gfCNCPoint4[7267] = {X 587.5052, Y 48.1018, Z -5.5000, A 0.000, B 0.000, C 0.000 }
gfCNCPoint4[7268] = {X 587.0658, Y 48.8401, Z -5.5000, A 0.000, B 0.000, C 0.000 }
gfCNCPoint4[7269] = {X 586.5368, Y 49.5171, Z -5.5000, A 0.000, B 0.000, C 0.000 }
gfCNCPoint4[7270] = {X 585.9266, Y 50.1220, Z -5.5000, A 0.000, B 0.000, C 0.000 }
gfCNCPoint4[7271] = {X 585.1803, Y 50.6880, Z -5.5000, A 0.000, B 0.000, C 0.000 }
gfCNCPoint4[7272] = {X 584.3634, Y 51.1461, Z -5.5000, A 0.000, B 0.000, C 0.000 }
gfCNCPoint4[7273] = {X 583.3013, Y 51.5442, Z -5.5000, A 0.000, B 0.000, C 0.000 }
gfCNCPoint4[7274] = {X 582.1877, Y 51.7603, Z -5.5000, A 0.000, B 0.000, C 0.000 }
gfCNCPoint4[7275] = {X 581.0538, Y 51.7882, Z -5.5000, A 0.000, B 0.000, C 0.000 }
gfCNCPoint4[7276] = {X 579.9310, Y 51.6273, Z -5.5000, A 0.000, B 0.000, C 0.000 }
gfCNCPoint4[7277] = {X 578.8505, Y 51.2819, Z -5.5000, A 0.000, B 0.000, C 0.000 }
gfCNCPoint4[7278] = {X 577.8425, Y 50.7618, Z -5.5000, A 0.000, B 0.000, C 0.000 }
gfCNCPoint4[7279] = {X 576.9350, Y 50.0813, Z -5.5000, A 0.000, B 0.000, C 0.000 }
gfCNCPoint4[7280] = {X 576.3133, Y 49.4513, Z -5.5000, A 0.000, B 0.000, C 0.000 }
gfCNCPoint4[7281] = {X 575.7786, Y 48.7459, Z -5.5000, A 0.000, B 0.000, C 0.000 }
gfCNCPoint4[7282] = {X 575.3401, Y 47.9770, Z -5.5000, A 0.000, B 0.000, C 0.000 }
gfCNCPoint4[7283] = {X 574.9017, Y 48.7459, Z -5.5000, A 0.000, B 0.000, C 0.000 }
gfCNCPoint4[7284] = {X 574.3670, Y 49.4513, Z -5.5000, A 0.000, B 0.000, C 0.000 }
gfCNCPoint4[7285] = {X 573.7453, Y 50.0813, Z -5.5000, A 0.000, B 0.000, C 0.000 }
gfCNCPoint4[7286] = {X 572.7526, Y 50.8143, Z -5.5000, A 0.000, B 0.000, C 0.000 }
gfCNCPoint4[7287] = {X 571.6437, Y 51.3558, Z -5.5000, A 0.000, B 0.000, C 0.000 }
gfCNCPoint4[7288] = {X 570.4553, Y 51.6880, Z -5.5000, A 0.000, B 0.000, C 0.000 }
gfCNCPoint4[7289] = {X 569.2264, Y 51.8000, Z -5.5000, A 0.000, B 0.000, C 0.000 }
gfCNCPoint4[7290] = {X 562.4443, Y 51.8000, Z -5.5000, A 0.000, B 0.000, C 0.000 }
gfCNCPoint4[7291] = {X 561.2635, Y 51.6967, Z -5.5000, A 0.000, B 0.000, C 0.000 }
gfCNCPoint4[7292] = {X 560.1186, Y 51.3899, Z -5.5000, A 0.000, B 0.000, C 0.000 }
gfCNCPoint4[7293] = {X 559.0443, Y 50.8890, Z -5.5000, A 0.000, B 0.000, C 0.000 }
gfCNCPoint4[7294] = {X 558.0733, Y 50.2091, Z -5.5000, A 0.000, B 0.000, C 0.000 }
gfCNCPoint4[7295] = {X 557.2352, Y 49.3710, Z -5.5000, A 0.000, B 0.000, C 0.000 }
gfCNCPoint4[7296] = {X 556.5553, Y 48.4000, Z -5.5000, A 0.000, B 0.000, C 0.000 }
gfCNCPoint4[7297] = {X 556.0544, Y 47.3257, Z -5.5000, A 0.000, B 0.000, C 0.000 }
gfCNCPoint4[7298] = {X 555.7476, Y 46.1808, Z -5.5000, A 0.000, B 0.000, C 0.000 }
gfCNCPoint4[7299] = {X 555.6443, Y 45.0000, Z -5.5000, A 0.000, B 0.000, C 0.000 }
gfCNCPoint4[7300] = {X 555.6443, Y 44.0662, Z -5.5000, A 0.000, B 0.000, C 0.000 }
gfCNCPoint4[7301] = {X 555.7452, Y 42.9113, Z -5.5000, A 0.000, B 0.000, C 0.000 }
gfCNCPoint4[7302] = {X 556.0400, Y 41.7902, Z -5.5000, A 0.000, B 0.000, C 0.000 }
gfCNCPoint4[7303] = {X 556.5200, Y 40.7350, Z -5.5000, A 0.000, B 0.000, C 0.000 }
gfCNCPoint4[7304] = {X 557.1715, Y 39.7762, Z -5.5000, A 0.000, B 0.000, C 0.000 }
gfCNCPoint4[7305] = {X 557.1715, Y 10.2279, Z -5.5000, A 0.000, B 0.000, C 0.000 }
gfCNCPoint4[7306] = {X 556.5255, Y 9.2818, Z -5.5000, A 0.000, B 0.000, C 0.000 }
gfCNCPoint4[7307] = {X 556.0475, Y 8.2407, Z -5.5000, A 0.000, B 0.000, C 0.000 }
gfCNCPoint4[7308] = {X 555.7510, Y 7.1341, Z -5.5000, A 0.000, B 0.000, C 0.000 }
gfCNCPoint4[7309] = {X 555.6446, Y 5.9935, Z -5.5000, A 0.000, B 0.000, C 0.000 }
gfCNCPoint4[7310] = {X 555.6443, Y 5.0000, Z -5.5000, A 0.000, B 0.000, C 0.000 }
gfCNCPoint4[7311] = {X 555.6452, Y 4.8909, Z -5.5000, A 0.000, B 0.000, C 0.000 }
gfCNCPoint4[7312] = {X 555.6478, Y 4.7819, Z -5.5000, A 0.000, B 0.000, C 0.000 }
gfCNCPoint4[7313] = {X 555.8079, Y 3.5174, Z -5.5000, A 0.000, B 0.000, C 0.000 }
gfCNCPoint4[7314] = {X 556.2012, Y 2.3049, Z -5.5000, A 0.000, B 0.000, C 0.000 }
gfCNCPoint4[7315] = {X 358.2599, Y 2.3049, Z -5.5000, A 0.000, B 0.000, C 0.000 }
gfCNCPoint4[7316] = {X 360.1211, Y 3.4745, Z -5.5000, A 0.000, B 0.000, C 0.000 }
gfCNCPoint4[7317] = {X 361.8537, Y 4.8274, Z -5.5000, A 0.000, B 0.000, C 0.000 }
gfCNCPoint4[7318] = {X 363.4396, Y 6.3495, Z -5.5000, A 0.000, B 0.000, C 0.000 }
gfCNCPoint4[7319] = {X 363.8248, Y 6.7699, Z -5.5000, A 0.000, B 0.000, C 0.000 }
gfCNCPoint4[7320] = {X 364.1987, Y 7.2003, Z -5.5000, A 0.000, B 0.000, C 0.000 }
gfCNCPoint4[7321] = {X 365.5801, Y 8.9956, Z -5.5000, A 0.000, B 0.000, C 0.000 }
gfCNCPoint4[7322] = {X 366.7977, Y 10.9058, Z -5.5000, A 0.000, B 0.000, C 0.000 }
gfCNCPoint4[7323] = {X 367.8422, Y 12.9160, Z -5.5000, A 0.000, B 0.000, C 0.000 }
gfCNCPoint4[7324] = {X 368.7052, Y 15.0104, Z -5.5000, A 0.000, B 0.000, C 0.000 }
gfCNCPoint4[7325] = {X 369.3802, Y 17.1728, Z -5.5000, A 0.000, B 0.000, C 0.000 }
gfCNCPoint4[7326] = {X 369.8619, Y 19.3862, Z -5.5000, A 0.000, B 0.000, C 0.000 }
gfCNCPoint4[7327] = {X 370.1835, Y 21.6514, Z -5.5000, A 0.000, B 0.000, C 0.000 }
gfCNCPoint4[7328] = {X 370.3440, Y 23.9336, Z -5.5000, A 0.000, B 0.000, C 0.000 }
gfCNCPoint4[7329] = {X 370.3424, Y 26.2214, Z -5.5000, A 0.000, B 0.000, C 0.000 }
gfCNCPoint4[7330] = {X 370.1789, Y 28.5034, Z -5.5000, A 0.000, B 0.000, C 0.000 }
gfCNCPoint4[7331] = {X 369.8542, Y 30.7681, Z -5.5000, A 0.000, B 0.000, C 0.000 }
gfCNCPoint4[7332] = {X 369.3419, Y 33.0745, Z -5.5000, A 0.000, B 0.000, C 0.000 }
gfCNCPoint4[7333] = {X 368.6154, Y 35.3227, Z -5.5000, A 0.000, B 0.000, C 0.000 }
gfCNCPoint4[7334] = {X 367.6811, Y 37.4927, Z -5.5000, A 0.000, B 0.000, C 0.000 }
gfCNCPoint4[7335] = {X 366.5474, Y 39.5655, Z -5.5000, A 0.000, B 0.000, C 0.000 }
gfCNCPoint4[7336] = {X 365.2241, Y 41.5227, Z -5.5000, A 0.000, B 0.000, C 0.000 }
gfCNCPoint4[7337] = {X 363.7788, Y 43.2829, Z -5.5000, A 0.000, B 0.000, C 0.000 }
gfCNCPoint4[7338] = {X 362.1632, Y 44.8883, Z -5.5000, A 0.000, B 0.000, C 0.000 }
gfCNCPoint4[7339] = {X 360.3939, Y 46.3225, Z -5.5000, A 0.000, B 0.000, C 0.000 }
gfCNCPoint4[7340] = {X 358.4890, Y 47.5708, Z -5.5000, A 0.000, B 0.000, C 0.000 }
gfCNCPoint4[7341] = {X 356.4678, Y 48.6206, Z -5.5000, A 0.000, B 0.000, C 0.000 }
gfCNCPoint4[7342] = {X 354.6708, Y 49.3145, Z -5.5000, A 0.000, B 0.000, C 0.000 }
gfCNCPoint4[7343] = {X 352.8231, Y 49.8595, Z -5.5000, A 0.000, B 0.000, C 0.000 }
gfCNCPoint4[7344] = {X 350.9372, Y 50.2518, Z -5.5000, A 0.000, B 0.000, C 0.000 }
gfCNCPoint4[7345] = {X 349.0255, Y 50.4889, Z -5.5000, A 0.000, B 0.000, C 0.000 }
gfCNCPoint4[7346] = {X 347.1008, Y 50.5692, Z -5.5000, A 0.000, B 0.000, C 0.000 }
gfCNCPoint4[7347] = {X 344.9874, Y 50.5330, Z -5.5000, A 0.000, B 0.000, C 0.000 }
gfCNCPoint4[7348] = {X 342.8850, Y 50.3138, Z -5.5000, A 0.000, B 0.000, C 0.000 }
gfCNCPoint4[7349] = {X 340.8096, Y 49.9133, Z -5.5000, A 0.000, B 0.000, C 0.000 }
gfCNCPoint4[7350] = {X 338.7767, Y 49.3343, Z -5.5000, A 0.000, B 0.000, C 0.000 }
gfCNCPoint4[7351] = {X 336.8016, Y 48.5814, Z -5.5000, A 0.000, B 0.000, C 0.000 }
gfCNCPoint4[7352] = {X 334.8992, Y 47.6601, Z -5.5000, A 0.000, B 0.000, C 0.000 }
gfCNCPoint4[7353] = {X 333.3417, Y 46.7040, Z -5.5000, A 0.000, B 0.000, C 0.000 }
gfCNCPoint4[7354] = {X 331.8604, Y 45.6336, Z -5.5000, A 0.000, B 0.000, C 0.000 }
gfCNCPoint4[7355] = {X 330.4636, Y 44.4550, Z -5.5000, A 0.000, B 0.000, C 0.000 }
gfCNCPoint4[7356] = {X 329.4663, Y 44.4078, Z -5.5000, A 0.000, B 0.000, C 0.000 }
gfCNCPoint4[7357] = {X 328.4996, Y 44.1587, Z -5.5000, A 0.000, B 0.000, C 0.000 }
gfCNCPoint4[7358] = {X 327.6038, Y 43.7181, Z -5.5000, A 0.000, B 0.000, C 0.000 }
gfCNCPoint4[7359] = {X 326.8164, Y 43.1044, Z -5.5000, A 0.000, B 0.000, C 0.000 }
gfCNCPoint4[7360] = {X 326.1897, Y 42.4934, Z -5.5000, A 0.000, B 0.000, C 0.000 }
gfCNCPoint4[7361] = {X 325.5686, Y 41.7541, Z -5.5000, A 0.000, B 0.000, C 0.000 }
gfCNCPoint4[7362] = {X 325.1052, Y 40.9070, Z -5.5000, A 0.000, B 0.000, C 0.000 }
gfCNCPoint4[7363] = {X 324.8177, Y 39.9852, Z -5.5000, A 0.000, B 0.000, C 0.000 }
gfCNCPoint4[7364] = {X 324.7172, Y 39.0249, Z -5.5000, A 0.000, B 0.000, C 0.000 }
gfCNCPoint4[7365] = {X 324.8079, Y 38.0635, Z -5.5000, A 0.000, B 0.000, C 0.000 }
gfCNCPoint4[7366] = {X 325.0860, Y 37.1389, Z -5.5000, A 0.000, B 0.000, C 0.000 }
gfCNCPoint4[7367] = {X 325.5408, Y 36.2871, Z -5.5000, A 0.000, B 0.000, C 0.000 }
gfCNCPoint4[7368] = {X 329.7765, Y 29.9537, Z -5.5000, A 0.000, B 0.000, C 0.000 }
gfCNCPoint4[7369] = {X 330.4614, Y 29.1399, Z -5.5000, A 0.000, B 0.000, C 0.000 }
gfCNCPoint4[7370] = {X 331.3063, Y 28.4938, Z -5.5000, A 0.000, B 0.000, C 0.000 }
gfCNCPoint4[7371] = {X 332.2712, Y 28.0462, Z -5.5000, A 0.000, B 0.000, C 0.000 }
gfCNCPoint4[7372] = {X 333.3101, Y 27.8182, Z -5.5000, A 0.000, B 0.000, C 0.000 }
gfCNCPoint4[7373] = {X 334.3737, Y 27.8207, Z -5.5000, A 0.000, B 0.000, C 0.000 }
gfCNCPoint4[7374] = {X 335.4116, Y 28.0536, Z -5.5000, A 0.000, B 0.000, C 0.000 }
gfCNCPoint4[7375] = {X 336.3743, Y 28.5058, Z -5.5000, A 0.000, B 0.000, C 0.000 }
gfCNCPoint4[7376] = {X 337.2161, Y 29.1559, Z -5.5000, A 0.000, B 0.000, C 0.000 }
gfCNCPoint4[7377] = {X 337.8209, Y 29.7388, Z -5.5000, A 0.000, B 0.000, C 0.000 }
gfCNCPoint4[7378] = {X 338.4993, Y 30.5708, Z -5.5000, A 0.000, B 0.000, C 0.000 }
gfCNCPoint4[7379] = {X 338.9793, Y 31.5311, Z -5.5000, A 0.000, B 0.000, C 0.000 }
gfCNCPoint4[7380] = {X 339.2378, Y 32.5730, Z -5.5000, A 0.000, B 0.000, C 0.000 }
gfCNCPoint4[7381] = {X 339.2621, Y 33.6463, Z -5.5000, A 0.000, B 0.000, C 0.000 }
gfCNCPoint4[7382] = {X 339.9099, Y 34.2186, Z -5.5000, A 0.000, B 0.000, C 0.000 }
gfCNCPoint4[7383] = {X 340.5785, Y 34.7664, Z -5.5000, A 0.000, B 0.000, C 0.000 }
gfCNCPoint4[7384] = {X 341.8101, Y 35.5739, Z -5.5000, A 0.000, B 0.000, C 0.000 }
gfCNCPoint4[7385] = {X 343.1464, Y 36.1929, Z -5.5000, A 0.000, B 0.000, C 0.000 }
gfCNCPoint4[7386] = {X 344.5587, Y 36.6102, Z -5.5000, A 0.000, B 0.000, C 0.000 }
gfCNCPoint4[7387] = {X 346.0168, Y 36.8169, Z -5.5000, A 0.000, B 0.000, C 0.000 }
gfCNCPoint4[7388] = {X 347.4895, Y 36.8085, Z -5.5000, A 0.000, B 0.000, C 0.000 }
gfCNCPoint4[7389] = {X 348.8389, Y 36.6273, Z -5.5000, A 0.000, B 0.000, C 0.000 }
gfCNCPoint4[7390] = {X 350.1409, Y 36.2289, Z -5.5000, A 0.000, B 0.000, C 0.000 }
gfCNCPoint4[7391] = {X 351.3606, Y 35.6237, Z -5.5000, A 0.000, B 0.000, C 0.000 }
gfCNCPoint4[7392] = {X 352.4655, Y 34.8281, Z -5.5000, A 0.000, B 0.000, C 0.000 }
gfCNCPoint4[7393] = {X 353.5665, Y 33.7584, Z -5.5000, A 0.000, B 0.000, C 0.000 }
gfCNCPoint4[7394] = {X 354.5195, Y 32.5548, Z -5.5000, A 0.000, B 0.000, C 0.000 }
gfCNCPoint4[7395] = {X 355.3081, Y 31.2377, Z -5.5000, A 0.000, B 0.000, C 0.000 }
gfCNCPoint4[7396] = {X 355.9192, Y 29.8294, Z -5.5000, A 0.000, B 0.000, C 0.000 }
gfCNCPoint4[7397] = {X 356.3423, Y 28.3537, Z -5.5000, A 0.000, B 0.000, C 0.000 }
gfCNCPoint4[7398] = {X 356.6068, Y 26.7185, Z -5.5000, A 0.000, B 0.000, C 0.000 }
gfCNCPoint4[7399] = {X 356.7145, Y 25.0656, Z -5.5000, A 0.000, B 0.000, C 0.000 }
gfCNCPoint4[7400] = {X 356.6644, Y 23.4100, Z -5.5000, A 0.000, B 0.000, C 0.000 }
gfCNCPoint4[7401] = {X 356.4569, Y 21.7666, Z -5.5000, A 0.000, B 0.000, C 0.000 }
gfCNCPoint4[7402] = {X 356.1201, Y 20.3209, Z -5.5000, A 0.000, B 0.000, C 0.000 }
gfCNCPoint4[7403] = {X 355.5964, Y 18.9319, Z -5.5000, A 0.000, B 0.000, C 0.000 }
gfCNCPoint4[7404] = {X 354.8948, Y 17.6237, Z -5.5000, A 0.000, B 0.000, C 0.000 }
gfCNCPoint4[7405] = {X 354.0275, Y 16.4190, Z -5.5000, A 0.000, B 0.000, C 0.000 }
gfCNCPoint4[7406] = {X 353.2099, Y 15.5481, Z -5.5000, A 0.000, B 0.000, C 0.000 }
gfCNCPoint4[7407] = {X 352.2795, Y 14.7991, Z -5.5000, A 0.000, B 0.000, C 0.000 }
gfCNCPoint4[7408] = {X 351.2542, Y 14.1863, Z -5.5000, A 0.000, B 0.000, C 0.000 }
gfCNCPoint4[7409] = {X 350.1538, Y 13.7217, Z -5.5000, A 0.000, B 0.000, C 0.000 }
gfCNCPoint4[7410] = {X 348.9995, Y 13.4142, Z -5.5000, A 0.000, B 0.000, C 0.000 }
gfCNCPoint4[7411] = {X 347.3622, Y 13.2074, Z -5.5000, A 0.000, B 0.000, C 0.000 }
gfCNCPoint4[7412] = {X 345.7118, Y 13.2126, Z -5.5000, A 0.000, B 0.000, C 0.000 }
gfCNCPoint4[7413] = {X 344.0758, Y 13.4298, Z -5.5000, A 0.000, B 0.000, C 0.000 }
gfCNCPoint4[7414] = {X 342.4812, Y 13.8553, Z -5.5000, A 0.000, B 0.000, C 0.000 }
gfCNCPoint4[7415] = {X 340.9545, Y 14.4821, Z -5.5000, A 0.000, B 0.000, C 0.000 }
gfCNCPoint4[7416] = {X 339.5209, Y 15.2999, Z -5.5000, A 0.000, B 0.000, C 0.000 }
gfCNCPoint4[7417] = {X 339.4271, Y 16.1855, Z -5.5000, A 0.000, B 0.000, C 0.000 }
gfCNCPoint4[7418] = {X 339.1739, Y 17.0393, Z -5.5000, A 0.000, B 0.000, C 0.000 }
gfCNCPoint4[7419] = {X 338.7698, Y 17.8330, Z -5.5000, A 0.000, B 0.000, C 0.000 }
gfCNCPoint4[7420] = {X 338.2281, Y 18.5399, Z -5.5000, A 0.000, B 0.000, C 0.000 }
gfCNCPoint4[7421] = {X 337.5670, Y 19.1366, Z -5.5000, A 0.000, B 0.000, C 0.000 }
gfCNCPoint4[7422] = {X 336.8400, Y 19.6716, Z -5.5000, A 0.000, B 0.000, C 0.000 }
gfCNCPoint4[7423] = {X 335.9171, Y 20.1909, Z -5.5000, A 0.000, B 0.000, C 0.000 }
gfCNCPoint4[7424] = {X 334.9039, Y 20.4988, Z -5.5000, A 0.000, B 0.000, C 0.000 }
gfCNCPoint4[7425] = {X 333.8481, Y 20.5809, Z -5.5000, A 0.000, B 0.000, C 0.000 }
gfCNCPoint4[7426] = {X 332.7995, Y 20.4334, Z -5.5000, A 0.000, B 0.000, C 0.000 }
gfCNCPoint4[7427] = {X 331.8074, Y 20.0631, Z -5.5000, A 0.000, B 0.000, C 0.000 }
gfCNCPoint4[7428] = {X 330.9186, Y 19.4875, Z -5.5000, A 0.000, B 0.000, C 0.000 }
gfCNCPoint4[7429] = {X 330.1748, Y 18.7338, Z -5.5000, A 0.000, B 0.000, C 0.000 }
gfCNCPoint4[7430] = {X 329.6111, Y 17.8373, Z -5.5000, A 0.000, B 0.000, C 0.000 }
gfCNCPoint4[7431] = {X 326.0906, Y 10.5950, Z -5.5000, A 0.000, B 0.000, C 0.000 }
gfCNCPoint4[7432] = {X 325.7555, Y 9.6856, Z -5.5000, A 0.000, B 0.000, C 0.000 }
gfCNCPoint4[7433] = {X 325.6067, Y 8.7279, Z -5.5000, A 0.000, B 0.000, C 0.000 }
gfCNCPoint4[7434] = {X 325.6502, Y 7.7597, Z -5.5000, A 0.000, B 0.000, C 0.000 }
gfCNCPoint4[7435] = {X 325.8842, Y 6.8191, Z -5.5000, A 0.000, B 0.000, C 0.000 }
gfCNCPoint4[7436] = {X 326.2994, Y 5.9434, Z -5.5000, A 0.000, B 0.000, C 0.000 }
gfCNCPoint4[7437] = {X 326.9295, Y 5.1131, Z -5.5000, A 0.000, B 0.000, C 0.000 }
gfCNCPoint4[7438] = {X 327.7216, Y 4.4356, Z -5.5000, A 0.000, B 0.000, C 0.000 }
gfCNCPoint4[7439] = {X 328.3967, Y 3.9733, Z -5.5000, A 0.000, B 0.000, C 0.000 }
gfCNCPoint4[7440] = {X 329.3293, Y 3.4828, Z -5.5000, A 0.000, B 0.000, C 0.000 }
gfCNCPoint4[7441] = {X 330.3454, Y 3.2040, Z -5.5000, A 0.000, B 0.000, C 0.000 }
gfCNCPoint4[7442] = {X 331.3977, Y 3.1498, Z -5.5000, A 0.000, B 0.000, C 0.000 }
gfCNCPoint4[7443] = {X 332.4371, Y 3.3227, Z -5.5000, A 0.000, B 0.000, C 0.000 }
gfCNCPoint4[7444] = {X 333.3743, Y 2.7962, Z -5.5000, A 0.000, B 0.000, C 0.000 }
gfCNCPoint4[7445] = {X 334.3304, Y 2.3049, Z -5.5000, A 0.000, B 0.000, C 0.000 }
gfCNCPoint4[7446] = {X 334.5418, Y 2.7359, Z -5.5000, A 0.000, B 0.000, C 0.000 }
gfCNCPoint4[7447] = {X 335.0189, Y 2.5073, Z -5.5000, A 0.000, B 0.000, C 0.000 }
gfCNCPoint4[7448] = {X 335.5002, Y 2.2876, Z -5.5000, A 0.000, B 0.000, C 0.000 }
gfCNCPoint4[7449] = {X 335.8480, Y 2.1328, Z -5.5000, A 0.000, B 0.000, C 0.000 }
gfCNCPoint4[7450] = {X 337.9512, Y 1.3123, Z -5.5000, A 0.000, B 0.000, C 0.000 }
gfCNCPoint4[7451] = {X 340.1169, Y 0.6747, Z -5.5000, A 0.000, B 0.000, C 0.000 }
gfCNCPoint4[7452] = {X 342.3292, Y 0.2248, Z -5.5000, A 0.000, B 0.000, C 0.000 }
gfCNCPoint4[7453] = {X 344.5719, Y -0.0341, Z -5.5000, A 0.000, B 0.000, C 0.000 }
gfCNCPoint4[7454] = {X 346.8285, Y -0.1003, Z -5.5000, A 0.000, B 0.000, C 0.000 }
gfCNCPoint4[7455] = {X 349.0825, Y 0.0269, Z -5.5000, A 0.000, B 0.000, C 0.000 }
gfCNCPoint4[7456] = {X 351.3173, Y 0.3465, Z -5.5000, A 0.000, B 0.000, C 0.000 }
gfCNCPoint4[7457] = {X 351.8883, Y 0.4533, Z -5.5000, A 0.000, B 0.000, C 0.000 }
gfCNCPoint4[7458] = {X 353.8461, Y 0.9459, Z -5.5000, A 0.000, B 0.000, C 0.000 }
gfCNCPoint4[7459] = {X 355.7478, Y 1.6233, Z -5.5000, A 0.000, B 0.000, C 0.000 }
gfCNCPoint4[7460] = {X 357.5760, Y 2.4795, Z -5.5000, A 0.000, B 0.000, C 0.000 }
gfCNCPoint4[7461] = {X 359.3141, Y 3.5064, Z -5.5000, A 0.000, B 0.000, C 0.000 }
gfCNCPoint4[7462] = {X 360.9460, Y 4.6948, Z -5.5000, A 0.000, B 0.000, C 0.000 }
gfCNCPoint4[7463] = {X 362.4569, Y 6.0337, Z -5.5000, A 0.000, B 0.000, C 0.000 }
gfCNCPoint4[7464] = {X 363.8328, Y 7.5110, Z -5.5000, A 0.000, B 0.000, C 0.000 }
gfCNCPoint4[7465] = {X 365.1882, Y 9.2728, Z -5.5000, A 0.000, B 0.000, C 0.000 }
gfCNCPoint4[7466] = {X 366.3829, Y 11.1473, Z -5.5000, A 0.000, B 0.000, C 0.000 }
gfCNCPoint4[7467] = {X 367.4076, Y 13.1198, Z -5.5000, A 0.000, B 0.000, C 0.000 }
gfCNCPoint4[7468] = {X 368.2544, Y 15.1751, Z -5.5000, A 0.000, B 0.000, C 0.000 }
gfCNCPoint4[7469] = {X 368.9166, Y 17.2970, Z -5.5000, A 0.000, B 0.000, C 0.000 }
gfCNCPoint4[7470] = {X 369.3891, Y 19.4690, Z -5.5000, A 0.000, B 0.000, C 0.000 }
gfCNCPoint4[7471] = {X 369.7061, Y 21.7011, Z -5.5000, A 0.000, B 0.000, C 0.000 }
gfCNCPoint4[7472] = {X 369.8643, Y 23.9499, Z -5.5000, A 0.000, B 0.000, C 0.000 }
gfCNCPoint4[7473] = {X 369.8628, Y 26.2044, Z -5.5000, A 0.000, B 0.000, C 0.000 }
gfCNCPoint4[7474] = {X 369.7016, Y 28.4531, Z -5.5000, A 0.000, B 0.000, C 0.000 }
gfCNCPoint4[7475] = {X 369.3815, Y 30.6847, Z -5.5000, A 0.000, B 0.000, C 0.000 }
gfCNCPoint4[7476] = {X 368.8789, Y 32.9479, Z -5.5000, A 0.000, B 0.000, C 0.000 }
gfCNCPoint4[7477] = {X 368.1661, Y 35.1539, Z -5.5000, A 0.000, B 0.000, C 0.000 }
gfCNCPoint4[7478] = {X 367.2493, Y 37.2832, Z -5.5000, A 0.000, B 0.000, C 0.000 }
gfCNCPoint4[7479] = {X 366.1366, Y 39.3171, Z -5.5000, A 0.000, B 0.000, C 0.000 }
gfCNCPoint4[7480] = {X 364.8380, Y 41.2375, Z -5.5000, A 0.000, B 0.000, C 0.000 }
gfCNCPoint4[7481] = {X 364.7204, Y 41.3984, Z -5.5000, A 0.000, B 0.000, C 0.000 }
gfCNCPoint4[7482] = {X 363.4201, Y 42.9672, Z -5.5000, A 0.000, B 0.000, C 0.000 }
gfCNCPoint4[7483] = {X 361.9805, Y 44.4093, Z -5.5000, A 0.000, B 0.000, C 0.000 }
gfCNCPoint4[7484] = {X 360.4141, Y 45.7125, Z -5.5000, A 0.000, B 0.000, C 0.000 }
gfCNCPoint4[7485] = {X 358.7341, Y 46.8657, Z -5.5000, A 0.000, B 0.000, C 0.000 }
gfCNCPoint4[7486] = {X 356.9549, Y 47.8589, Z -5.5000, A 0.000, B 0.000, C 0.000 }
gfCNCPoint4[7487] = {X 356.2499, Y 48.1924, Z -5.5000, A 0.000, B 0.000, C 0.000 }
gfCNCPoint4[7488] = {X 354.0456, Y 49.0148, Z -5.5000, A 0.000, B 0.000, C 0.000 }
gfCNCPoint4[7489] = {X 351.7691, Y 49.6088, Z -5.5000, A 0.000, B 0.000, C 0.000 }
gfCNCPoint4[7490] = {X 349.4440, Y 49.9682, Z -5.5000, A 0.000, B 0.000, C 0.000 }
gfCNCPoint4[7491] = {X 347.0943, Y 50.0893, Z -5.5000, A 0.000, B 0.000, C 0.000 }
gfCNCPoint4[7492] = {X 345.0202, Y 50.0541, Z -5.5000, A 0.000, B 0.000, C 0.000 }
gfCNCPoint4[7493] = {X 342.9570, Y 49.8392, Z -5.5000, A 0.000, B 0.000, C 0.000 }
gfCNCPoint4[7494] = {X 340.9201, Y 49.4461, Z -5.5000, A 0.000, B 0.000, C 0.000 }
gfCNCPoint4[7495] = {X 338.9251, Y 48.8778, Z -5.5000, A 0.000, B 0.000, C 0.000 }
gfCNCPoint4[7496] = {X 336.9869, Y 48.1385, Z -5.5000, A 0.000, B 0.000, C 0.000 }
gfCNCPoint4[7497] = {X 335.1201, Y 47.2339, Z -5.5000, A 0.000, B 0.000, C 0.000 }
gfCNCPoint4[7498] = {X 333.5415, Y 46.2602, Z -5.5000, A 0.000, B 0.000, C 0.000 }
gfCNCPoint4[7499] = {X 332.0433, Y 45.1668, Z -5.5000, A 0.000, B 0.000, C 0.000 }
gfCNCPoint4[7500] = {X 330.6345, Y 43.9603, Z -5.5000, A 0.000, B 0.000, C 0.000 }
gfCNCPoint4[7501] = {X 329.6760, Y 43.9518, Z -5.5000, A 0.000, B 0.000, C 0.000 }
gfCNCPoint4[7502] = {X 328.7420, Y 43.7358, Z -5.5000, A 0.000, B 0.000, C 0.000 }
gfCNCPoint4[7503] = {X 327.8770, Y 43.3228, Z -5.5000, A 0.000, B 0.000, C 0.000 }
gfCNCPoint4[7504] = {X 327.1220, Y 42.7321, Z -5.5000, A 0.000, B 0.000, C 0.000 }
gfCNCPoint4[7505] = {X 326.5249, Y 42.1498, Z -5.5000, A 0.000, B 0.000, C 0.000 }
gfCNCPoint4[7506] = {X 325.8848, Y 41.3619, Z -5.5000, A 0.000, B 0.000, C 0.000 }
gfCNCPoint4[7507] = {X 325.4424, Y 40.4483, Z -5.5000, A 0.000, B 0.000, C 0.000 }
gfCNCPoint4[7508] = {X 325.2210, Y 39.4576, Z -5.5000, A 0.000, B 0.000, C 0.000 }
gfCNCPoint4[7509] = {X 325.2326, Y 38.4426, Z -5.5000, A 0.000, B 0.000, C 0.000 }
gfCNCPoint4[7510] = {X 325.4765, Y 37.4572, Z -5.5000, A 0.000, B 0.000, C 0.000 }
gfCNCPoint4[7511] = {X 325.9397, Y 36.5539, Z -5.5000, A 0.000, B 0.000, C 0.000 }
gfCNCPoint4[7512] = {X 330.1988, Y 30.1861, Z -5.5000, A 0.000, B 0.000, C 0.000 }
gfCNCPoint4[7513] = {X 330.8195, Y 29.4619, Z -5.5000, A 0.000, B 0.000, C 0.000 }
gfCNCPoint4[7514] = {X 331.5816, Y 28.8884, Z -5.5000, A 0.000, B 0.000, C 0.000 }
gfCNCPoint4[7515] = {X 332.4495, Y 28.4927, Z -5.5000, A 0.000, B 0.000, C 0.000 }
gfCNCPoint4[7516] = {X 333.3822, Y 28.2932, Z -5.5000, A 0.000, B 0.000, C 0.000 }
gfCNCPoint4[7517] = {X 334.3360, Y 28.2995, Z -5.5000, A 0.000, B 0.000, C 0.000 }
gfCNCPoint4[7518] = {X 335.2660, Y 28.5111, Z -5.5000, A 0.000, B 0.000, C 0.000 }
gfCNCPoint4[7519] = {X 336.1286, Y 28.9182, Z -5.5000, A 0.000, B 0.000, C 0.000 }
gfCNCPoint4[7520] = {X 336.8831, Y 29.5016, Z -5.5000, A 0.000, B 0.000, C 0.000 }
gfCNCPoint4[7521] = {X 337.4845, Y 30.0811, Z -5.5000, A 0.000, B 0.000, C 0.000 }
gfCNCPoint4[7522] = {X 338.1271, Y 30.8800, Z -5.5000, A 0.000, B 0.000, C 0.000 }
gfCNCPoint4[7523] = {X 338.5674, Y 31.8058, Z -5.5000, A 0.000, B 0.000, C 0.000 }
gfCNCPoint4[7524] = {X 338.7815, Y 32.8084, Z -5.5000, A 0.000, B 0.000, C 0.000 }
gfCNCPoint4[7525] = {X 338.7578, Y 33.8333, Z -5.5000, A 0.000, B 0.000, C 0.000 }
gfCNCPoint4[7526] = {X 339.5070, Y 34.5056, Z -5.5000, A 0.000, B 0.000, C 0.000 }
gfCNCPoint4[7527] = {X 340.2840, Y 35.1455, Z -5.5000, A 0.000, B 0.000, C 0.000 }
gfCNCPoint4[7528] = {X 341.4952, Y 35.9470, Z -5.5000, A 0.000, B 0.000, C 0.000 }
gfCNCPoint4[7529] = {X 342.8050, Y 36.5744, Z -5.5000, A 0.000, B 0.000, C 0.000 }
gfCNCPoint4[7530] = {X 344.1886, Y 37.0158, Z -5.5000, A 0.000, B 0.000, C 0.000 }
gfCNCPoint4[7531] = {X 345.6198, Y 37.2628, Z -5.5000, A 0.000, B 0.000, C 0.000 }
gfCNCPoint4[7532] = {X 347.0713, Y 37.3108, Z -5.5000, A 0.000, B 0.000, C 0.000 }
gfCNCPoint4[7533] = {X 347.5143, Y 37.2879, Z -5.5000, A 0.000, B 0.000, C 0.000 }
gfCNCPoint4[7534] = {X 348.9415, Y 37.0963, Z -5.5000, A 0.000, B 0.000, C 0.000 }
gfCNCPoint4[7535] = {X 350.3184, Y 36.6748, Z -5.5000, A 0.000, B 0.000, C 0.000 }
gfCNCPoint4[7536] = {X 351.6083, Y 36.0348, Z -5.5000, A 0.000, B 0.000, C 0.000 }
gfCNCPoint4[7537] = {X 352.7768, Y 35.1934, Z -5.5000, A 0.000, B 0.000, C 0.000 }
gfCNCPoint4[7538] = {X 353.9229, Y 34.0800, Z -5.5000, A 0.000, B 0.000, C 0.000 }
gfCNCPoint4[7539] = {X 354.9147, Y 32.8272, Z -5.5000, A 0.000, B 0.000, C 0.000 }
gfCNCPoint4[7540] = {X 355.7355, Y 31.4562, Z -5.5000, A 0.000, B 0.000, C 0.000 }
gfCNCPoint4[7541] = {X 356.3714, Y 29.9903, Z -5.5000, A 0.000, B 0.000, C 0.000 }
gfCNCPoint4[7542] = {X 356.8116, Y 28.4543, Z -5.5000, A 0.000, B 0.000, C 0.000 }
gfCNCPoint4[7543] = {X 357.0837, Y 26.7727, Z -5.5000, A 0.000, B 0.000, C 0.000 }
gfCNCPoint4[7544] = {X 357.1944, Y 25.0729, Z -5.5000, A 0.000, B 0.000, C 0.000 }
gfCNCPoint4[7545] = {X 357.1427, Y 23.3702, Z -5.5000, A 0.000, B 0.000, C 0.000 }
gfCNCPoint4[7546] = {X 356.9291, Y 21.6802, Z -5.5000, A 0.000, B 0.000, C 0.000 }
gfCNCPoint4[7547] = {X 356.5774, Y 20.1748, Z -5.5000, A 0.000, B 0.000, C 0.000 }
gfCNCPoint4[7548] = {X 356.0312, Y 18.7285, Z -5.5000, A 0.000, B 0.000, C 0.000 }
gfCNCPoint4[7549] = {X 355.3000, Y 17.3664, Z -5.5000, A 0.000, B 0.000, C 0.000 }
gfCNCPoint4[7550] = {X 354.3964, Y 16.1120, Z -5.5000, A 0.000, B 0.000, C 0.000 }
gfCNCPoint4[7551] = {X 353.5334, Y 15.1935, Z -5.5000, A 0.000, B 0.000, C 0.000 }
gfCNCPoint4[7552] = {X 352.5515, Y 14.4035, Z -5.5000, A 0.000, B 0.000, C 0.000 }
gfCNCPoint4[7553] = {X 351.4695, Y 13.7573, Z -5.5000, A 0.000, B 0.000, C 0.000 }
gfCNCPoint4[7554] = {X 350.3084, Y 13.2673, Z -5.5000, A 0.000, B 0.000, C 0.000 }
gfCNCPoint4[7555] = {X 349.0905, Y 12.9429, Z -5.5000, A 0.000, B 0.000, C 0.000 }
gfCNCPoint4[7556] = {X 347.3478, Y 12.7257, Z -5.5000, A 0.000, B 0.000, C 0.000 }
gfCNCPoint4[7557] = {X 345.5917, Y 12.7399, Z -5.5000, A 0.000, B 0.000, C 0.000 }
gfCNCPoint4[7558] = {X 343.8528, Y 12.9854, Z -5.5000, A 0.000, B 0.000, C 0.000 }
gfCNCPoint4[7559] = {X 342.1614, Y 13.4578, Z -5.5000, A 0.000, B 0.000, C 0.000 }
gfCNCPoint4[7560] = {X 340.5469, Y 14.1489, Z -5.5000, A 0.000, B 0.000, C 0.000 }
gfCNCPoint4[7561] = {X 339.0376, Y 15.0467, Z -5.5000, A 0.000, B 0.000, C 0.000 }
gfCNCPoint4[7562] = {X 338.9895, Y 15.9046, Z -5.5000, A 0.000, B 0.000, C 0.000 }
gfCNCPoint4[7563] = {X 338.7757, Y 16.7367, Z -5.5000, A 0.000, B 0.000, C 0.000 }
gfCNCPoint4[7564] = {X 338.4042, Y 17.5115, Z -5.5000, A 0.000, B 0.000, C 0.000 }
gfCNCPoint4[7565] = {X 337.8892, Y 18.1992, Z -5.5000, A 0.000, B 0.000, C 0.000 }
gfCNCPoint4[7566] = {X 337.2504, Y 18.7738, Z -5.5000, A 0.000, B 0.000, C 0.000 }
gfCNCPoint4[7567] = {X 336.5606, Y 19.2813, Z -5.5000, A 0.000, B 0.000, C 0.000 }
gfCNCPoint4[7568] = {X 335.7284, Y 19.7495, Z -5.5000, A 0.000, B 0.000, C 0.000 }
gfCNCPoint4[7569] = {X 334.8148, Y 20.0271, Z -5.5000, A 0.000, B 0.000, C 0.000 }
gfCNCPoint4[7570] = {X 333.8628, Y 20.1012, Z -5.5000, A 0.000, B 0.000, C 0.000 }
gfCNCPoint4[7571] = {X 332.9173, Y 19.9681, Z -5.5000, A 0.000, B 0.000, C 0.000 }
gfCNCPoint4[7572] = {X 332.0228, Y 19.6341, Z -5.5000, A 0.000, B 0.000, C 0.000 }
gfCNCPoint4[7573] = {X 331.2213, Y 19.1151, Z -5.5000, A 0.000, B 0.000, C 0.000 }
gfCNCPoint4[7574] = {X 330.5507, Y 18.4353, Z -5.5000, A 0.000, B 0.000, C 0.000 }
gfCNCPoint4[7575] = {X 330.0425, Y 17.6269, Z -5.5000, A 0.000, B 0.000, C 0.000 }
gfCNCPoint4[7576] = {X 326.5223, Y 10.3852, Z -5.5000, A 0.000, B 0.000, C 0.000 }
gfCNCPoint4[7577] = {X 326.2154, Y 9.5469, Z -5.5000, A 0.000, B 0.000, C 0.000 }
gfCNCPoint4[7578] = {X 326.0841, Y 8.6639, Z -5.5000, A 0.000, B 0.000, C 0.000 }
gfCNCPoint4[7579] = {X 326.1338, Y 7.7725, Z -5.5000, A 0.000, B 0.000, C 0.000 }
gfCNCPoint4[7580] = {X 326.3623, Y 6.9096, Z -5.5000, A 0.000, B 0.000, C 0.000 }
gfCNCPoint4[7581] = {X 326.7603, Y 6.1105, Z -5.5000, A 0.000, B 0.000, C 0.000 }
gfCNCPoint4[7582] = {X 327.3114, Y 5.4082, Z -5.5000, A 0.000, B 0.000, C 0.000 }
gfCNCPoint4[7583] = {X 327.9929, Y 4.8316, Z -5.5000, A 0.000, B 0.000, C 0.000 }
gfCNCPoint4[7584] = {X 328.6647, Y 4.3715, Z -5.5000, A 0.000, B 0.000, C 0.000 }
gfCNCPoint4[7585] = {X 329.5523, Y 3.9112, Z -5.5000, A 0.000, B 0.000, C 0.000 }
gfCNCPoint4[7586] = {X 330.5209, Y 3.6631, Z -5.5000, A 0.000, B 0.000, C 0.000 }
gfCNCPoint4[7587] = {X 331.5205, Y 3.6401, Z -5.5000, A 0.000, B 0.000, C 0.000 }
gfCNCPoint4[7588] = {X 332.4995, Y 3.8435, Z -5.5000, A 0.000, B 0.000, C 0.000 }
gfCNCPoint4[7589] = {X 333.5093, Y 3.2688, Z -5.5000, A 0.000, B 0.000, C 0.000 }
gfCNCPoint4[7590] = {X 334.5418, Y 2.7359, Z -5.5000, A 0.000, B 0.000, C 0.000 }
gfCNCPoint4[7591] = {X 334.3304, Y 2.3049, Z -5.5000, A 0.000, B 0.000, C 0.000 }
gfCNCPoint4[7592] = {X 2.3034, Y 2.3049, Z -5.5000, A 0.000, B 0.000, C 0.000 }
gfCNCPoint4[7593] = {X 2.3034, Y 6.8597, Z -5.5000, A 0.000, B 0.000, C 0.000 }
gfCNCPoint4[7594] = {X 2.3913, Y 6.8772, Z -5.5000, A 0.000, B 0.000, C 0.000 }
gfCNCPoint4[7595] = {X 2.8672, Y 6.6841, Z -5.5000, A 0.000, B 0.000, C 0.000 }
gfCNCPoint4[7596] = {X 3.3507, Y 6.5108, Z -5.5000, A 0.000, B 0.000, C 0.000 }
gfCNCPoint4[7597] = {X 5.4534, Y 5.7817, Z -5.5000, A 0.000, B 0.000, C 0.000 }
gfCNCPoint4[7598] = {X 7.6109, Y 5.2354, Z -5.5000, A 0.000, B 0.000, C 0.000 }
gfCNCPoint4[7599] = {X 9.8072, Y 4.8761, Z -5.5000, A 0.000, B 0.000, C 0.000 }
gfCNCPoint4[7600] = {X 12.0263, Y 4.7063, Z -5.5000, A 0.000, B 0.000, C 0.000 }
gfCNCPoint4[7601] = {X 14.2517, Y 4.7273, Z -5.5000, A 0.000, B 0.000, C 0.000 }
gfCNCPoint4[7602] = {X 16.4672, Y 4.9389, Z -5.5000, A 0.000, B 0.000, C 0.000 }
gfCNCPoint4[7603] = {X 18.0967, Y 5.2197, Z -5.5000, A 0.000, B 0.000, C 0.000 }
gfCNCPoint4[7604] = {X 19.6973, Y 5.6345, Z -5.5000, A 0.000, B 0.000, C 0.000 }
gfCNCPoint4[7605] = {X 21.2581, Y 6.1807, Z -5.5000, A 0.000, B 0.000, C 0.000 }
gfCNCPoint4[7606] = {X 22.7682, Y 6.8543, Z -5.5000, A 0.000, B 0.000, C 0.000 }
gfCNCPoint4[7607] = {X 24.4890, Y 7.8182, Z -5.5000, A 0.000, B 0.000, C 0.000 }
gfCNCPoint4[7608] = {X 26.1061, Y 8.9475, Z -5.5000, A 0.000, B 0.000, C 0.000 }
gfCNCPoint4[7609] = {X 27.4003, Y 10.0777, Z -5.5000, A 0.000, B 0.000, C 0.000 }
gfCNCPoint4[7610] = {X 28.5613, Y 11.3445, Z -5.5000, A 0.000, B 0.000, C 0.000 }
gfCNCPoint4[7611] = {X 29.5748, Y 12.7321, Z -5.5000, A 0.000, B 0.000, C 0.000 }
gfCNCPoint4[7612] = {X 30.4282, Y 14.2235, Z -5.5000, A 0.000, B 0.000, C 0.000 }
gfCNCPoint4[7613] = {X 31.1110, Y 15.8003, Z -5.5000, A 0.000, B 0.000, C 0.000 }
gfCNCPoint4[7614] = {X 31.6708, Y 17.7360, Z -5.5000, A 0.000, B 0.000, C 0.000 }
gfCNCPoint4[7615] = {X 32.0041, Y 19.7232, Z -5.5000, A 0.000, B 0.000, C 0.000 }
gfCNCPoint4[7616] = {X 32.1064, Y 21.7356, Z -5.5000, A 0.000, B 0.000, C 0.000 }
gfCNCPoint4[7617] = {X 31.9764, Y 23.7464, Z -5.5000, A 0.000, B 0.000, C 0.000 }
gfCNCPoint4[7618] = {X 31.6157, Y 25.7289, Z -5.5000, A 0.000, B 0.000, C 0.000 }
gfCNCPoint4[7619] = {X 31.1968, Y 27.1578, Z -5.5000, A 0.000, B 0.000, C 0.000 }
gfCNCPoint4[7620] = {X 30.6302, Y 28.5349, Z -5.5000, A 0.000, B 0.000, C 0.000 }
gfCNCPoint4[7621] = {X 29.9223, Y 29.8450, Z -5.5000, A 0.000, B 0.000, C 0.000 }
gfCNCPoint4[7622] = {X 29.0808, Y 31.0735, Z -5.5000, A 0.000, B 0.000, C 0.000 }
gfCNCPoint4[7623] = {X 29.6385, Y 31.7918, Z -5.5000, A 0.000, B 0.000, C 0.000 }
gfCNCPoint4[7624] = {X 30.0953, Y 32.5782, Z -5.5000, A 0.000, B 0.000, C 0.000 }
gfCNCPoint4[7625] = {X 33.1423, Y 38.8726, Z -5.5000, A 0.000, B 0.000, C 0.000 }
gfCNCPoint4[7626] = {X 33.5391, Y 39.8957, Z -5.5000, A 0.000, B 0.000, C 0.000 }
gfCNCPoint4[7627] = {X 33.7662, Y 40.9694, Z -5.5000, A 0.000, B 0.000, C 0.000 }
gfCNCPoint4[7628] = {X 33.8177, Y 42.0656, Z -5.5000, A 0.000, B 0.000, C 0.000 }
gfCNCPoint4[7629] = {X 33.7164, Y 43.0266, Z -5.5000, A 0.000, B 0.000, C 0.000 }
gfCNCPoint4[7630] = {X 33.4799, Y 43.9636, Z -5.5000, A 0.000, B 0.000, C 0.000 }
gfCNCPoint4[7631] = {X 33.1103, Y 44.8630, Z -5.5000, A 0.000, B 0.000, C 0.000 }
gfCNCPoint4[7632] = {X 32.6161, Y 45.7005, Z -5.5000, A 0.000, B 0.000, C 0.000 }
gfCNCPoint4[7633] = {X 32.0075, Y 46.4590, Z -5.5000, A 0.000, B 0.000, C 0.000 }
gfCNCPoint4[7634] = {X 31.2970, Y 47.1229, Z -5.5000, A 0.000, B 0.000, C 0.000 }
gfCNCPoint4[7635] = {X 30.7604, Y 47.5568, Z -5.5000, A 0.000, B 0.000, C 0.000 }
gfCNCPoint4[7636] = {X 29.8545, Y 48.1753, Z -5.5000, A 0.000, B 0.000, C 0.000 }
gfCNCPoint4[7637] = {X 28.8611, Y 48.6405, Z -5.5000, A 0.000, B 0.000, C 0.000 }
gfCNCPoint4[7638] = {X 27.8060, Y 48.9401, Z -5.5000, A 0.000, B 0.000, C 0.000 }
gfCNCPoint4[7639] = {X 26.7164, Y 49.0666, Z -5.5000, A 0.000, B 0.000, C 0.000 }
gfCNCPoint4[7640] = {X 25.6207, Y 49.0165, Z -5.5000, A 0.000, B 0.000, C 0.000 }
gfCNCPoint4[7641] = {X 23.9304, Y 49.8556, Z -5.5000, A 0.000, B 0.000, C 0.000 }
gfCNCPoint4[7642] = {X 22.1931, Y 50.5925, Z -5.5000, A 0.000, B 0.000, C 0.000 }
gfCNCPoint4[7643] = {X 20.4150, Y 51.2246, Z -5.5000, A 0.000, B 0.000, C 0.000 }
gfCNCPoint4[7644] = {X 18.2656, Y 51.8305, Z -5.5000, A 0.000, B 0.000, C 0.000 }
gfCNCPoint4[7645] = {X 16.0711, Y 52.2441, Z -5.5000, A 0.000, B 0.000, C 0.000 }
gfCNCPoint4[7646] = {X 13.8486, Y 52.4621, Z -5.5000, A 0.000, B 0.000, C 0.000 }
gfCNCPoint4[7647] = {X 11.6155, Y 52.4828, Z -5.5000, A 0.000, B 0.000, C 0.000 }
gfCNCPoint4[7648] = {X 9.3893, Y 52.3061, Z -5.5000, A 0.000, B 0.000, C 0.000 }
gfCNCPoint4[7649] = {X 7.1875, Y 51.9334, Z -5.5000, A 0.000, B 0.000, C 0.000 }
gfCNCPoint4[7650] = {X 6.2988, Y 51.7232, Z -5.5000, A 0.000, B 0.000, C 0.000 }
gfCNCPoint4[7651] = {X 5.4211, Y 51.4710, Z -5.5000, A 0.000, B 0.000, C 0.000 }
gfCNCPoint4[7652] = {X 3.8339, Y 50.8957, Z -5.5000, A 0.000, B 0.000, C 0.000 }
gfCNCPoint4[7653] = {X 2.3034, Y 50.1830, Z -5.5000, A 0.000, B 0.000, C 0.000 }
gfCNCPoint4[7654] = {X 2.3034, Y 97.6951, Z -5.5000, A 0.000, B 0.000, C 0.000 }
gfCNCPoint4[7655] = {X 120.1200, Y 97.6951, Z -5.5000, A 0.000, B 0.000, C 0.000 }
gfCNCPoint4[7656] = {X 120.1200, Y 97.0659, Z -5.5000, A 0.000, B 0.000, C 0.000 }
gfCNCPoint4[7657] = {X 120.2338, Y 96.0183, Z -5.5000, A 0.000, B 0.000, C 0.000 }
gfCNCPoint4[7658] = {X 120.5698, Y 95.0195, Z -5.5000, A 0.000, B 0.000, C 0.000 }
gfCNCPoint4[7659] = {X 121.1124, Y 94.1161, Z -5.5000, A 0.000, B 0.000, C 0.000 }
gfCNCPoint4[7660] = {X 121.8364, Y 93.3503, Z -5.5000, A 0.000, B 0.000, C 0.000 }
gfCNCPoint4[7661] = {X 122.7078, Y 92.7578, Z -5.5000, A 0.000, B 0.000, C 0.000 }
gfCNCPoint4[7662] = {X 123.6861, Y 92.3661, Z -5.5000, A 0.000, B 0.000, C 0.000 }
gfCNCPoint4[7663] = {X 124.7257, Y 92.1936, Z -5.5000, A 0.000, B 0.000, C 0.000 }
gfCNCPoint4[7664] = {X 124.7852, Y 92.1783, Z -5.5000, A 0.000, B 0.000, C 0.000 }
gfCNCPoint4[7665] = {X 124.8456, Y 92.1672, Z -5.5000, A 0.000, B 0.000, C 0.000 }
gfCNCPoint4[7666] = {X 125.3649, Y 92.0902, Z -5.5000, A 0.000, B 0.000, C 0.000 }
gfCNCPoint4[7667] = {X 126.0997, Y 91.9691, Z -5.5000, A 0.000, B 0.000, C 0.000 }
gfCNCPoint4[7668] = {X 126.8254, Y 91.8017, Z -5.5000, A 0.000, B 0.000, C 0.000 }
gfCNCPoint4[7669] = {X 127.9732, Y 90.7128, Z -5.5000, A 0.000, B 0.000, C 0.000 }
gfCNCPoint4[7670] = {X 129.0625, Y 89.5654, Z -5.5000, A 0.000, B 0.000, C 0.000 }
gfCNCPoint4[7671] = {X 154.9459, Y 61.1418, Z -5.5000, A 0.000, B 0.000, C 0.000 }
gfCNCPoint4[7672] = {X 154.6592, Y 60.4493, Z -5.5000, A 0.000, B 0.000, C 0.000 }
gfCNCPoint4[7673] = {X 154.4818, Y 59.7211, Z -5.5000, A 0.000, B 0.000, C 0.000 }
gfCNCPoint4[7674] = {X 154.4181, Y 58.9744, Z -5.5000, A 0.000, B 0.000, C 0.000 }
gfCNCPoint4[7675] = {X 154.4180, Y 58.0000, Z -5.5000, A 0.000, B 0.000, C 0.000 }
gfCNCPoint4[7676] = {X 154.5117, Y 57.0480, Z -5.5000, A 0.000, B 0.000, C 0.000 }
gfCNCPoint4[7677] = {X 154.7894, Y 56.1325, Z -5.5000, A 0.000, B 0.000, C 0.000 }
gfCNCPoint4[7678] = {X 155.2404, Y 55.2888, Z -5.5000, A 0.000, B 0.000, C 0.000 }
gfCNCPoint4[7679] = {X 155.8473, Y 54.5493, Z -5.5000, A 0.000, B 0.000, C 0.000 }
gfCNCPoint4[7680] = {X 156.5868, Y 53.9424, Z -5.5000, A 0.000, B 0.000, C 0.000 }
gfCNCPoint4[7681] = {X 157.4305, Y 53.4915, Z -5.5000, A 0.000, B 0.000, C 0.000 }
gfCNCPoint4[7682] = {X 158.3459, Y 53.2138, Z -5.5000, A 0.000, B 0.000, C 0.000 }
gfCNCPoint4[7683] = {X 159.2980, Y 53.1200, Z -5.5000, A 0.000, B 0.000, C 0.000 }
gfCNCPoint4[7684] = {X 178.5335, Y 53.1200, Z -5.5000, A 0.000, B 0.000, C 0.000 }
gfCNCPoint4[7685] = {X 179.4855, Y 53.2138, Z -5.5000, A 0.000, B 0.000, C 0.000 }
gfCNCPoint4[7686] = {X 180.4010, Y 53.4915, Z -5.5000, A 0.000, B 0.000, C 0.000 }
gfCNCPoint4[7687] = {X 181.2447, Y 53.9424, Z -5.5000, A 0.000, B 0.000, C 0.000 }
gfCNCPoint4[7688] = {X 181.9842, Y 54.5493, Z -5.5000, A 0.000, B 0.000, C 0.000 }
gfCNCPoint4[7689] = {X 182.5911, Y 55.2888, Z -5.5000, A 0.000, B 0.000, C 0.000 }
gfCNCPoint4[7690] = {X 183.0420, Y 56.1325, Z -5.5000, A 0.000, B 0.000, C 0.000 }
gfCNCPoint4[7691] = {X 183.3197, Y 57.0480, Z -5.5000, A 0.000, B 0.000, C 0.000 }
gfCNCPoint4[7692] = {X 183.4135, Y 58.0000, Z -5.5000, A 0.000, B 0.000, C 0.000 }
gfCNCPoint4[7693] = {X 183.4133, Y 58.9744, Z -5.5000, A 0.000, B 0.000, C 0.000 }
gfCNCPoint4[7694] = {X 183.3512, Y 59.7111, Z -5.5000, A 0.000, B 0.000, C 0.000 }
gfCNCPoint4[7695] = {X 183.1785, Y 60.4301, Z -5.5000, A 0.000, B 0.000, C 0.000 }
gfCNCPoint4[7696] = {X 182.8992, Y 61.1147, Z -5.5000, A 0.000, B 0.000, C 0.000 }
gfCNCPoint4[7697] = {X 209.8921, Y 90.5759, Z -5.5000, A 0.000, B 0.000, C 0.000 }
gfCNCPoint4[7698] = {X 210.5202, Y 91.2133, Z -5.5000, A 0.000, B 0.000, C 0.000 }
gfCNCPoint4[7699] = {X 211.1931, Y 91.8031, Z -5.5000, A 0.000, B 0.000, C 0.000 }
gfCNCPoint4[7700] = {X 211.3594, Y 91.9077, Z -5.5000, A 0.000, B 0.000, C 0.000 }
gfCNCPoint4[7701] = {X 211.5460, Y 91.9689, Z -5.5000, A 0.000, B 0.000, C 0.000 }
gfCNCPoint4[7702] = {X 212.2018, Y 92.1091, Z -5.5000, A 0.000, B 0.000, C 0.000 }
gfCNCPoint4[7703] = {X 213.4084, Y 92.2611, Z -5.5000, A 0.000, B 0.000, C 0.000 }
gfCNCPoint4[7704] = {X 214.4425, Y 92.1749, Z -5.5000, A 0.000, B 0.000, C 0.000 }
gfCNCPoint4[7705] = {X 215.4785, Y 92.1160, Z -5.5000, A 0.000, B 0.000, C 0.000 }
gfCNCPoint4[7706] = {X 216.0525, Y 92.0563, Z -5.5000, A 0.000, B 0.000, C 0.000 }
gfCNCPoint4[7707] = {X 216.6053, Y 91.8910, Z -5.5000, A 0.000, B 0.000, C 0.000 }
gfCNCPoint4[7708] = {X 217.1179, Y 91.6259, Z -5.5000, A 0.000, B 0.000, C 0.000 }
gfCNCPoint4[7709] = {X 244.6006, Y 74.0196, Z -5.5000, A 0.000, B 0.000, C 0.000 }
gfCNCPoint4[7710] = {X 221.4278, Y 64.9261, Z -5.5000, A 0.000, B 0.000, C 0.000 }
gfCNCPoint4[7711] = {X 219.7199, Y 64.3539, Z -5.5000, A 0.000, B 0.000, C 0.000 }
gfCNCPoint4[7712] = {X 217.9578, Y 63.9806, Z -5.5000, A 0.000, B 0.000, C 0.000 }
gfCNCPoint4[7713] = {X 216.1645, Y 63.8112, Z -5.5000, A 0.000, B 0.000, C 0.000 }
gfCNCPoint4[7714] = {X 215.1120, Y 63.6594, Z -5.5000, A 0.000, B 0.000, C 0.000 }
gfCNCPoint4[7715] = {X 214.1173, Y 63.2832, Z -5.5000, A 0.000, B 0.000, C 0.000 }
gfCNCPoint4[7716] = {X 213.2278, Y 62.7004, Z -5.5000, A 0.000, B 0.000, C 0.000 }
gfCNCPoint4[7717] = {X 212.4856, Y 61.9388, Z -5.5000, A 0.000, B 0.000, C 0.000 }
gfCNCPoint4[7718] = {X 211.9260, Y 61.0345, Z -5.5000, A 0.000, B 0.000, C 0.000 }
gfCNCPoint4[7719] = {X 211.5756, Y 60.0305, Z -5.5000, A 0.000, B 0.000, C 0.000 }
gfCNCPoint4[7720] = {X 211.4510, Y 58.9744, Z -5.5000, A 0.000, B 0.000, C 0.000 }
gfCNCPoint4[7721] = {X 211.4508, Y 58.0000, Z -5.5000, A 0.000, B 0.000, C 0.000 }
gfCNCPoint4[7722] = {X 211.5446, Y 57.0480, Z -5.5000, A 0.000, B 0.000, C 0.000 }
gfCNCPoint4[7723] = {X 211.8223, Y 56.1325, Z -5.5000, A 0.000, B 0.000, C 0.000 }
gfCNCPoint4[7724] = {X 212.2732, Y 55.2888, Z -5.5000, A 0.000, B 0.000, C 0.000 }
gfCNCPoint4[7725] = {X 212.8801, Y 54.5493, Z -5.5000, A 0.000, B 0.000, C 0.000 }
gfCNCPoint4[7726] = {X 213.6196, Y 53.9424, Z -5.5000, A 0.000, B 0.000, C 0.000 }
gfCNCPoint4[7727] = {X 214.4633, Y 53.4915, Z -5.5000, A 0.000, B 0.000, C 0.000 }
gfCNCPoint4[7728] = {X 215.3788, Y 53.2138, Z -5.5000, A 0.000, B 0.000, C 0.000 }
gfCNCPoint4[7729] = {X 216.3308, Y 53.1200, Z -5.5000, A 0.000, B 0.000, C 0.000 }
gfCNCPoint4[7730] = {X 237.2617, Y 53.1200, Z -5.5000, A 0.000, B 0.000, C 0.000 }
gfCNCPoint4[7731] = {X 238.3265, Y 53.2376, Z -5.5000, A 0.000, B 0.000, C 0.000 }
gfCNCPoint4[7732] = {X 239.3400, Y 53.5847, Z -5.5000, A 0.000, B 0.000, C 0.000 }
gfCNCPoint4[7733] = {X 240.2533, Y 54.1445, Z -5.5000, A 0.000, B 0.000, C 0.000 }
gfCNCPoint4[7734] = {X 241.0224, Y 54.8902, Z -5.5000, A 0.000, B 0.000, C 0.000 }
gfCNCPoint4[7735] = {X 241.6104, Y 55.7857, Z -5.5000, A 0.000, B 0.000, C 0.000 }
gfCNCPoint4[7736] = {X 241.9888, Y 56.7879, Z -5.5000, A 0.000, B 0.000, C 0.000 }
gfCNCPoint4[7737] = {X 242.1393, Y 57.8485, Z -5.5000, A 0.000, B 0.000, C 0.000 }
gfCNCPoint4[7738] = {X 248.3217, Y 60.2592, Z -5.5000, A 0.000, B 0.000, C 0.000 }
gfCNCPoint4[7739] = {X 275.0724, Y 70.8770, Z -5.5000, A 0.000, B 0.000, C 0.000 }
gfCNCPoint4[7740] = {X 275.0721, Y 63.6740, Z -5.5000, A 0.000, B 0.000, C 0.000 }
gfCNCPoint4[7741] = {X 274.0639, Y 63.3056, Z -5.5000, A 0.000, B 0.000, C 0.000 }
gfCNCPoint4[7742] = {X 273.1606, Y 62.7257, Z -5.5000, A 0.000, B 0.000, C 0.000 }
gfCNCPoint4[7743] = {X 272.4060, Y 61.9624, Z -5.5000, A 0.000, B 0.000, C 0.000 }
gfCNCPoint4[7744] = {X 271.8365, Y 61.0526, Z -5.5000, A 0.000, B 0.000, C 0.000 }
gfCNCPoint4[7745] = {X 271.4797, Y 60.0402, Z -5.5000, A 0.000, B 0.000, C 0.000 }
gfCNCPoint4[7746] = {X 271.3529, Y 58.9744, Z -5.5000, A 0.000, B 0.000, C 0.000 }
gfCNCPoint4[7747] = {X 271.3527, Y 58.0000, Z -5.5000, A 0.000, B 0.000, C 0.000 }
gfCNCPoint4[7748] = {X 271.4465, Y 57.0480, Z -5.5000, A 0.000, B 0.000, C 0.000 }
gfCNCPoint4[7749] = {X 271.7242, Y 56.1325, Z -5.5000, A 0.000, B 0.000, C 0.000 }
gfCNCPoint4[7750] = {X 272.1751, Y 55.2888, Z -5.5000, A 0.000, B 0.000, C 0.000 }
gfCNCPoint4[7751] = {X 272.7820, Y 54.5493, Z -5.5000, A 0.000, B 0.000, C 0.000 }
gfCNCPoint4[7752] = {X 273.5215, Y 53.9424, Z -5.5000, A 0.000, B 0.000, C 0.000 }
gfCNCPoint4[7753] = {X 274.3652, Y 53.4915, Z -5.5000, A 0.000, B 0.000, C 0.000 }
gfCNCPoint4[7754] = {X 275.2806, Y 53.2138, Z -5.5000, A 0.000, B 0.000, C 0.000 }
gfCNCPoint4[7755] = {X 276.2327, Y 53.1200, Z -5.5000, A 0.000, B 0.000, C 0.000 }
gfCNCPoint4[7756] = {X 292.7731, Y 53.1200, Z -5.5000, A 0.000, B 0.000, C 0.000 }
gfCNCPoint4[7757] = {X 293.7251, Y 53.2138, Z -5.5000, A 0.000, B 0.000, C 0.000 }
gfCNCPoint4[7758] = {X 294.6406, Y 53.4915, Z -5.5000, A 0.000, B 0.000, C 0.000 }
gfCNCPoint4[7759] = {X 295.4843, Y 53.9424, Z -5.5000, A 0.000, B 0.000, C 0.000 }
gfCNCPoint4[7760] = {X 296.2238, Y 54.5493, Z -5.5000, A 0.000, B 0.000, C 0.000 }
gfCNCPoint4[7761] = {X 296.8307, Y 55.2888, Z -5.5000, A 0.000, B 0.000, C 0.000 }
gfCNCPoint4[7762] = {X 297.2816, Y 56.1325, Z -5.5000, A 0.000, B 0.000, C 0.000 }
gfCNCPoint4[7763] = {X 297.5593, Y 57.0480, Z -5.5000, A 0.000, B 0.000, C 0.000 }
gfCNCPoint4[7764] = {X 297.6531, Y 58.0000, Z -5.5000, A 0.000, B 0.000, C 0.000 }
gfCNCPoint4[7765] = {X 297.6531, Y 58.9367, Z -5.5000, A 0.000, B 0.000, C 0.000 }
gfCNCPoint4[7766] = {X 297.5309, Y 60.0090, Z -5.5000, A 0.000, B 0.000, C 0.000 }
gfCNCPoint4[7767] = {X 297.1768, Y 61.0285, Z -5.5000, A 0.000, B 0.000, C 0.000 }
gfCNCPoint4[7768] = {X 296.6080, Y 61.9456, Z -5.5000, A 0.000, B 0.000, C 0.000 }
gfCNCPoint4[7769] = {X 295.8521, Y 62.7159, Z -5.5000, A 0.000, B 0.000, C 0.000 }
gfCNCPoint4[7770] = {X 294.9458, Y 63.3018, Z -5.5000, A 0.000, B 0.000, C 0.000 }
gfCNCPoint4[7771] = {X 293.9331, Y 63.6750, Z -5.5000, A 0.000, B 0.000, C 0.000 }
gfCNCPoint4[7772] = {X 293.9331, Y 92.3198, Z -5.5000, A 0.000, B 0.000, C 0.000 }
gfCNCPoint4[7773] = {X 294.9449, Y 92.6952, Z -5.5000, A 0.000, B 0.000, C 0.000 }
gfCNCPoint4[7774] = {X 295.8504, Y 93.2825, Z -5.5000, A 0.000, B 0.000, C 0.000 }
gfCNCPoint4[7775] = {X 296.6057, Y 94.0533, Z -5.5000, A 0.000, B 0.000, C 0.000 }
gfCNCPoint4[7776] = {X 297.1745, Y 94.9705, Z -5.5000, A 0.000, B 0.000, C 0.000 }
gfCNCPoint4[7777] = {X 297.5294, Y 95.9897, Z -5.5000, A 0.000, B 0.000, C 0.000 }
gfCNCPoint4[7778] = {X 297.6531, Y 97.0618, Z -5.5000, A 0.000, B 0.000, C 0.000 }
gfCNCPoint4[7779] = {X 297.6531, Y 97.6951, Z -5.5000, A 0.000, B 0.000, C 0.000 }
gfCNCPoint4[7780] = {X 297.1731, Y 97.6951, Z -5.5000, A 0.000, B 0.000, C 0.000 }
gfCNCPoint4[7781] = {X 297.1731, Y 98.0000, Z -5.5000, A 0.000, B 0.000, C 0.000 }
gfCNCPoint4[7782] = {X 297.0628, Y 98.9791, Z -5.5000, A 0.000, B 0.000, C 0.000 }
gfCNCPoint4[7783] = {X 296.7373, Y 99.9091, Z -5.5000, A 0.000, B 0.000, C 0.000 }
gfCNCPoint4[7784] = {X 296.2131, Y 100.7434, Z -5.5000, A 0.000, B 0.000, C 0.000 }
gfCNCPoint4[7785] = {X 295.5164, Y 101.4401, Z -5.5000, A 0.000, B 0.000, C 0.000 }
gfCNCPoint4[7786] = {X 294.6822, Y 101.9643, Z -5.5000, A 0.000, B 0.000, C 0.000 }
gfCNCPoint4[7787] = {X 293.7522, Y 102.2897, Z -5.5000, A 0.000, B 0.000, C 0.000 }
gfCNCPoint4[7788] = {X 292.7731, Y 102.4000, Z -5.5000, A 0.000, B 0.000, C 0.000 }
gfCNCPoint4[7789] = {X 276.2327, Y 102.4000, Z -5.5000, A 0.000, B 0.000, C 0.000 }
gfCNCPoint4[7790] = {X 275.2536, Y 102.2897, Z -5.5000, A 0.000, B 0.000, C 0.000 }
gfCNCPoint4[7791] = {X 274.3236, Y 101.9643, Z -5.5000, A 0.000, B 0.000, C 0.000 }
gfCNCPoint4[7792] = {X 273.4893, Y 101.4401, Z -5.5000, A 0.000, B 0.000, C 0.000 }
gfCNCPoint4[7793] = {X 272.7926, Y 100.7434, Z -5.5000, A 0.000, B 0.000, C 0.000 }
gfCNCPoint4[7794] = {X 272.2684, Y 99.9091, Z -5.5000, A 0.000, B 0.000, C 0.000 }
gfCNCPoint4[7795] = {X 271.9430, Y 98.9791, Z -5.5000, A 0.000, B 0.000, C 0.000 }
gfCNCPoint4[7796] = {X 271.8327, Y 98.0000, Z -5.5000, A 0.000, B 0.000, C 0.000 }
gfCNCPoint4[7797] = {X 271.8329, Y 97.0190, Z -5.5000, A 0.000, B 0.000, C 0.000 }
gfCNCPoint4[7798] = {X 271.9305, Y 96.1432, Z -5.5000, A 0.000, B 0.000, C 0.000 }
gfCNCPoint4[7799] = {X 272.2006, Y 95.3045, Z -5.5000, A 0.000, B 0.000, C 0.000 }
gfCNCPoint4[7800] = {X 272.6325, Y 94.5364, Z -5.5000, A 0.000, B 0.000, C 0.000 }
gfCNCPoint4[7801] = {X 273.2087, Y 93.8698, Z -5.5000, A 0.000, B 0.000, C 0.000 }
gfCNCPoint4[7802] = {X 273.9062, Y 93.3313, Z -5.5000, A 0.000, B 0.000, C 0.000 }
gfCNCPoint4[7803] = {X 274.6970, Y 92.9426, Z -5.5000, A 0.000, B 0.000, C 0.000 }
gfCNCPoint4[7804] = {X 275.5494, Y 92.7193, Z -5.5000, A 0.000, B 0.000, C 0.000 }
gfCNCPoint4[7805] = {X 275.5494, Y 85.6495, Z -5.5000, A 0.000, B 0.000, C 0.000 }
gfCNCPoint4[7806] = {X 262.6482, Y 80.5923, Z -5.5000, A 0.000, B 0.000, C 0.000 }
gfCNCPoint4[7807] = {X 262.3205, Y 80.7990, Z -5.5000, A 0.000, B 0.000, C 0.000 }
gfCNCPoint4[7808] = {X 237.8772, Y 96.6315, Z -5.5000, A 0.000, B 0.000, C 0.000 }
gfCNCPoint4[7809] = {X 237.8798, Y 97.0659, Z -5.5000, A 0.000, B 0.000, C 0.000 }
gfCNCPoint4[7810] = {X 237.8798, Y 98.0000, Z -5.5000, A 0.000, B 0.000, C 0.000 }
gfCNCPoint4[7811] = {X 237.7695, Y 98.9791, Z -5.5000, A 0.000, B 0.000, C 0.000 }
gfCNCPoint4[7812] = {X 237.4440, Y 99.9091, Z -5.5000, A 0.000, B 0.000, C 0.000 }
gfCNCPoint4[7813] = {X 236.9198, Y 100.7434, Z -5.5000, A 0.000, B 0.000, C 0.000 }
gfCNCPoint4[7814] = {X 236.2231, Y 101.4401, Z -5.5000, A 0.000, B 0.000, C 0.000 }
gfCNCPoint4[7815] = {X 235.3889, Y 101.9643, Z -5.5000, A 0.000, B 0.000, C 0.000 }
gfCNCPoint4[7816] = {X 234.4589, Y 102.2897, Z -5.5000, A 0.000, B 0.000, C 0.000 }
gfCNCPoint4[7817] = {X 233.4798, Y 102.4000, Z -5.5000, A 0.000, B 0.000, C 0.000 }
gfCNCPoint4[7818] = {X 214.1790, Y 102.4000, Z -5.5000, A 0.000, B 0.000, C 0.000 }
gfCNCPoint4[7819] = {X 213.7862, Y 102.3824, Z -5.5000, A 0.000, B 0.000, C 0.000 }
gfCNCPoint4[7820] = {X 213.3966, Y 102.3299, Z -5.5000, A 0.000, B 0.000, C 0.000 }
gfCNCPoint4[7821] = {X 213.0069, Y 102.3824, Z -5.5000, A 0.000, B 0.000, C 0.000 }
gfCNCPoint4[7822] = {X 212.6141, Y 102.4000, Z -5.5000, A 0.000, B 0.000, C 0.000 }
gfCNCPoint4[7823] = {X 194.9870, Y 102.4000, Z -5.5000, A 0.000, B 0.000, C 0.000 }
gfCNCPoint4[7824] = {X 194.0079, Y 102.2897, Z -5.5000, A 0.000, B 0.000, C 0.000 }
gfCNCPoint4[7825] = {X 193.0779, Y 101.9643, Z -5.5000, A 0.000, B 0.000, C 0.000 }
gfCNCPoint4[7826] = {X 192.2436, Y 101.4401, Z -5.5000, A 0.000, B 0.000, C 0.000 }
gfCNCPoint4[7827] = {X 191.5469, Y 100.7434, Z -5.5000, A 0.000, B 0.000, C 0.000 }
gfCNCPoint4[7828] = {X 191.0227, Y 99.9091, Z -5.5000, A 0.000, B 0.000, C 0.000 }
gfCNCPoint4[7829] = {X 190.6973, Y 98.9791, Z -5.5000, A 0.000, B 0.000, C 0.000 }
gfCNCPoint4[7830] = {X 190.5870, Y 98.0000, Z -5.5000, A 0.000, B 0.000, C 0.000 }
gfCNCPoint4[7831] = {X 190.5870, Y 97.0659, Z -5.5000, A 0.000, B 0.000, C 0.000 }
gfCNCPoint4[7832] = {X 190.6897, Y 96.1207, Z -5.5000, A 0.000, B 0.000, C 0.000 }
gfCNCPoint4[7833] = {X 190.9931, Y 95.2196, Z -5.5000, A 0.000, B 0.000, C 0.000 }
gfCNCPoint4[7834] = {X 191.4830, Y 94.4047, Z -5.5000, A 0.000, B 0.000, C 0.000 }
gfCNCPoint4[7835] = {X 188.5295, Y 91.1802, Z -5.5000, A 0.000, B 0.000, C 0.000 }
gfCNCPoint4[7836] = {X 150.1254, Y 91.1802, Z -5.5000, A 0.000, B 0.000, C 0.000 }
gfCNCPoint4[7837] = {X 147.2498, Y 94.3661, Z -5.5000, A 0.000, B 0.000, C 0.000 }
gfCNCPoint4[7838] = {X 147.7557, Y 95.1904, Z -5.5000, A 0.000, B 0.000, C 0.000 }
gfCNCPoint4[7839] = {X 148.0705, Y 96.1049, Z -5.5000, A 0.000, B 0.000, C 0.000 }
gfCNCPoint4[7840] = {X 148.1791, Y 97.0661, Z -5.5000, A 0.000, B 0.000, C 0.000 }
gfCNCPoint4[7841] = {X 148.1791, Y 98.0000, Z -5.5000, A 0.000, B 0.000, C 0.000 }
gfCNCPoint4[7842] = {X 148.0688, Y 98.9791, Z -5.5000, A 0.000, B 0.000, C 0.000 }
gfCNCPoint4[7843] = {X 147.7434, Y 99.9091, Z -5.5000, A 0.000, B 0.000, C 0.000 }
gfCNCPoint4[7844] = {X 147.2192, Y 100.7434, Z -5.5000, A 0.000, B 0.000, C 0.000 }
gfCNCPoint4[7845] = {X 146.5225, Y 101.4401, Z -5.5000, A 0.000, B 0.000, C 0.000 }
gfCNCPoint4[7846] = {X 145.6882, Y 101.9643, Z -5.5000, A 0.000, B 0.000, C 0.000 }
gfCNCPoint4[7847] = {X 144.7582, Y 102.2897, Z -5.5000, A 0.000, B 0.000, C 0.000 }
gfCNCPoint4[7848] = {X 143.7791, Y 102.4000, Z -5.5000, A 0.000, B 0.000, C 0.000 }
gfCNCPoint4[7849] = {X 125.0000, Y 102.4000, Z -5.5000, A 0.000, B 0.000, C 0.000 }
gfCNCPoint4[7850] = {X 124.0209, Y 102.2897, Z -5.5000, A 0.000, B 0.000, C 0.000 }
gfCNCPoint4[7851] = {X 123.0909, Y 101.9643, Z -5.5000, A 0.000, B 0.000, C 0.000 }
gfCNCPoint4[7852] = {X 122.2566, Y 101.4401, Z -5.5000, A 0.000, B 0.000, C 0.000 }
gfCNCPoint4[7853] = {X 121.5599, Y 100.7434, Z -5.5000, A 0.000, B 0.000, C 0.000 }
gfCNCPoint4[7854] = {X 121.0357, Y 99.9091, Z -5.5000, A 0.000, B 0.000, C 0.000 }
gfCNCPoint4[7855] = {X 120.7103, Y 98.9791, Z -5.5000, A 0.000, B 0.000, C 0.000 }
gfCNCPoint4[7856] = {X 120.6000, Y 98.0000, Z -5.5000, A 0.000, B 0.000, C 0.000 }
gfCNCPoint4[7857] = {X 120.6000, Y 97.0659, Z -5.5000, A 0.000, B 0.000, C 0.000 }
gfCNCPoint4[7858] = {X 120.7046, Y 96.1122, Z -5.5000, A 0.000, B 0.000, C 0.000 }
gfCNCPoint4[7859] = {X 121.0134, Y 95.2039, Z -5.5000, A 0.000, B 0.000, C 0.000 }
gfCNCPoint4[7860] = {X 121.5118, Y 94.3840, Z -5.5000, A 0.000, B 0.000, C 0.000 }
gfCNCPoint4[7861] = {X 122.1761, Y 93.6917, Z -5.5000, A 0.000, B 0.000, C 0.000 }
gfCNCPoint4[7862] = {X 122.9746, Y 93.1598, Z -5.5000, A 0.000, B 0.000, C 0.000 }
gfCNCPoint4[7863] = {X 123.8694, Y 92.8137, Z -5.5000, A 0.000, B 0.000, C 0.000 }
gfCNCPoint4[7864] = {X 124.8179, Y 92.6697, Z -5.5000, A 0.000, B 0.000, C 0.000 }
gfCNCPoint4[7865] = {X 124.8661, Y 92.6527, Z -5.5000, A 0.000, B 0.000, C 0.000 }
gfCNCPoint4[7866] = {X 124.9161, Y 92.6420, Z -5.5000, A 0.000, B 0.000, C 0.000 }
gfCNCPoint4[7867] = {X 125.4412, Y 92.5641, Z -5.5000, A 0.000, B 0.000, C 0.000 }
gfCNCPoint4[7868] = {X 126.2565, Y 92.4272, Z -5.5000, A 0.000, B 0.000, C 0.000 }
gfCNCPoint4[7869] = {X 127.0607, Y 92.2354, Z -5.5000, A 0.000, B 0.000, C 0.000 }
gfCNCPoint4[7870] = {X 128.2724, Y 91.0923, Z -5.5000, A 0.000, B 0.000, C 0.000 }
gfCNCPoint4[7871] = {X 129.4203, Y 89.8854, Z -5.5000, A 0.000, B 0.000, C 0.000 }
gfCNCPoint4[7872] = {X 133.5081, Y 85.3888, Z -5.5000, A 0.000, B 0.000, C 0.000 }
gfCNCPoint4[7873] = {X 155.5326, Y 61.2105, Z -5.5000, A 0.000, B 0.000, C 0.000 }
gfCNCPoint4[7874] = {X 155.1839, Y 60.4944, Z -5.5000, A 0.000, B 0.000, C 0.000 }
gfCNCPoint4[7875] = {X 154.9700, Y 59.7272, Z -5.5000, A 0.000, B 0.000, C 0.000 }
gfCNCPoint4[7876] = {X 154.8980, Y 58.9341, Z -5.5000, A 0.000, B 0.000, C 0.000 }
gfCNCPoint4[7877] = {X 154.8980, Y 58.0000, Z -5.5000, A 0.000, B 0.000, C 0.000 }
gfCNCPoint4[7878] = {X 155.0083, Y 57.0209, Z -5.5000, A 0.000, B 0.000, C 0.000 }
gfCNCPoint4[7879] = {X 155.3337, Y 56.0909, Z -5.5000, A 0.000, B 0.000, C 0.000 }
gfCNCPoint4[7880] = {X 155.8579, Y 55.2566, Z -5.5000, A 0.000, B 0.000, C 0.000 }
gfCNCPoint4[7881] = {X 156.5546, Y 54.5599, Z -5.5000, A 0.000, B 0.000, C 0.000 }
gfCNCPoint4[7882] = {X 157.3889, Y 54.0357, Z -5.5000, A 0.000, B 0.000, C 0.000 }
gfCNCPoint4[7883] = {X 158.3189, Y 53.7103, Z -5.5000, A 0.000, B 0.000, C 0.000 }
gfCNCPoint4[7884] = {X 159.2980, Y 53.6000, Z -5.5000, A 0.000, B 0.000, C 0.000 }
gfCNCPoint4[7885] = {X 178.5335, Y 53.6000, Z -5.5000, A 0.000, B 0.000, C 0.000 }
gfCNCPoint4[7886] = {X 179.5126, Y 53.7103, Z -5.5000, A 0.000, B 0.000, C 0.000 }
gfCNCPoint4[7887] = {X 180.4426, Y 54.0357, Z -5.5000, A 0.000, B 0.000, C 0.000 }
gfCNCPoint4[7888] = {X 181.2769, Y 54.5599, Z -5.5000, A 0.000, B 0.000, C 0.000 }
gfCNCPoint4[7889] = {X 181.9736, Y 55.2566, Z -5.5000, A 0.000, B 0.000, C 0.000 }
gfCNCPoint4[7890] = {X 182.4978, Y 56.0909, Z -5.5000, A 0.000, B 0.000, C 0.000 }
gfCNCPoint4[7891] = {X 182.8232, Y 57.0209, Z -5.5000, A 0.000, B 0.000, C 0.000 }
gfCNCPoint4[7892] = {X 182.9335, Y 58.0000, Z -5.5000, A 0.000, B 0.000, C 0.000 }
gfCNCPoint4[7893] = {X 182.9334, Y 58.9704, Z -5.5000, A 0.000, B 0.000, C 0.000 }
gfCNCPoint4[7894] = {X 182.8587, Y 59.7417, Z -5.5000, A 0.000, B 0.000, C 0.000 }
gfCNCPoint4[7895] = {X 182.6500, Y 60.4879, Z -5.5000, A 0.000, B 0.000, C 0.000 }
gfCNCPoint4[7896] = {X 182.3136, Y 61.1860, Z -5.5000, A 0.000, B 0.000, C 0.000 }
gfCNCPoint4[7897] = {X 209.5382, Y 90.9002, Z -5.5000, A 0.000, B 0.000, C 0.000 }
gfCNCPoint4[7898] = {X 210.1909, Y 91.5624, Z -5.5000, A 0.000, B 0.000, C 0.000 }
gfCNCPoint4[7899] = {X 210.8900, Y 92.1754, Z -5.5000, A 0.000, B 0.000, C 0.000 }
gfCNCPoint4[7900] = {X 211.1519, Y 92.3405, Z -5.5000, A 0.000, B 0.000, C 0.000 }
gfCNCPoint4[7901] = {X 211.4457, Y 92.4383, Z -5.5000, A 0.000, B 0.000, C 0.000 }
gfCNCPoint4[7902] = {X 212.1215, Y 92.5828, Z -5.5000, A 0.000, B 0.000, C 0.000 }
gfCNCPoint4[7903] = {X 213.4015, Y 92.7441, Z -5.5000, A 0.000, B 0.000, C 0.000 }
gfCNCPoint4[7904] = {X 214.4548, Y 92.6553, Z -5.5000, A 0.000, B 0.000, C 0.000 }
gfCNCPoint4[7905] = {X 215.5100, Y 92.5952, Z -5.5000, A 0.000, B 0.000, C 0.000 }
gfCNCPoint4[7906] = {X 216.1640, Y 92.5232, Z -5.5000, A 0.000, B 0.000, C 0.000 }
gfCNCPoint4[7907] = {X 216.7937, Y 92.3325, Z -5.5000, A 0.000, B 0.000, C 0.000 }
gfCNCPoint4[7908] = {X 217.3777, Y 92.0295, Z -5.5000, A 0.000, B 0.000, C 0.000 }
gfCNCPoint4[7909] = {X 222.9188, Y 88.4535, Z -5.5000, A 0.000, B 0.000, C 0.000 }
gfCNCPoint4[7910] = {X 245.6525, Y 73.9167, Z -5.5000, A 0.000, B 0.000, C 0.000 }
gfCNCPoint4[7911] = {X 221.6009, Y 64.4783, Z -5.5000, A 0.000, B 0.000, C 0.000 }
gfCNCPoint4[7912] = {X 219.8422, Y 63.8897, Z -5.5000, A 0.000, B 0.000, C 0.000 }
gfCNCPoint4[7913] = {X 218.0279, Y 63.5057, Z -5.5000, A 0.000, B 0.000, C 0.000 }
gfCNCPoint4[7914] = {X 216.1816, Y 63.3315, Z -5.5000, A 0.000, B 0.000, C 0.000 }
gfCNCPoint4[7915] = {X 215.2274, Y 63.1935, Z -5.5000, A 0.000, B 0.000, C 0.000 }
gfCNCPoint4[7916] = {X 214.3262, Y 62.8509, Z -5.5000, A 0.000, B 0.000, C 0.000 }
gfCNCPoint4[7917] = {X 213.5213, Y 62.3203, Z -5.5000, A 0.000, B 0.000, C 0.000 }
gfCNCPoint4[7918] = {X 212.8512, Y 61.6271, Z -5.5000, A 0.000, B 0.000, C 0.000 }
gfCNCPoint4[7919] = {X 212.3482, Y 60.8046, Z -5.5000, A 0.000, B 0.000, C 0.000 }
gfCNCPoint4[7920] = {X 212.0364, Y 59.8923, Z -5.5000, A 0.000, B 0.000, C 0.000 }
gfCNCPoint4[7921] = {X 211.9308, Y 58.9341, Z -5.5000, A 0.000, B 0.000, C 0.000 }
gfCNCPoint4[7922] = {X 211.9308, Y 58.0000, Z -5.5000, A 0.000, B 0.000, C 0.000 }
gfCNCPoint4[7923] = {X 212.0411, Y 57.0209, Z -5.5000, A 0.000, B 0.000, C 0.000 }
gfCNCPoint4[7924] = {X 212.3665, Y 56.0909, Z -5.5000, A 0.000, B 0.000, C 0.000 }
gfCNCPoint4[7925] = {X 212.8907, Y 55.2566, Z -5.5000, A 0.000, B 0.000, C 0.000 }
gfCNCPoint4[7926] = {X 213.5875, Y 54.5599, Z -5.5000, A 0.000, B 0.000, C 0.000 }
gfCNCPoint4[7927] = {X 214.4217, Y 54.0357, Z -5.5000, A 0.000, B 0.000, C 0.000 }
gfCNCPoint4[7928] = {X 215.3517, Y 53.7103, Z -5.5000, A 0.000, B 0.000, C 0.000 }
gfCNCPoint4[7929] = {X 216.3308, Y 53.6000, Z -5.5000, A 0.000, B 0.000, C 0.000 }
gfCNCPoint4[7930] = {X 237.2617, Y 53.6000, Z -5.5000, A 0.000, B 0.000, C 0.000 }
gfCNCPoint4[7931] = {X 238.2408, Y 53.7103, Z -5.5000, A 0.000, B 0.000, C 0.000 }
gfCNCPoint4[7932] = {X 239.1708, Y 54.0357, Z -5.5000, A 0.000, B 0.000, C 0.000 }
gfCNCPoint4[7933] = {X 240.0050, Y 54.5599, Z -5.5000, A 0.000, B 0.000, C 0.000 }
gfCNCPoint4[7934] = {X 240.7017, Y 55.2566, Z -5.5000, A 0.000, B 0.000, C 0.000 }
gfCNCPoint4[7935] = {X 241.2260, Y 56.0909, Z -5.5000, A 0.000, B 0.000, C 0.000 }
gfCNCPoint4[7936] = {X 241.5514, Y 57.0209, Z -5.5000, A 0.000, B 0.000, C 0.000 }
gfCNCPoint4[7937] = {X 241.6617, Y 58.0000, Z -5.5000, A 0.000, B 0.000, C 0.000 }
gfCNCPoint4[7938] = {X 241.6617, Y 58.1774, Z -5.5000, A 0.000, B 0.000, C 0.000 }
gfCNCPoint4[7939] = {X 248.1446, Y 60.7053, Z -5.5000, A 0.000, B 0.000, C 0.000 }
gfCNCPoint4[7940] = {X 275.5525, Y 71.5840, Z -5.5000, A 0.000, B 0.000, C 0.000 }
gfCNCPoint4[7941] = {X 275.5520, Y 63.2811, Z -5.5000, A 0.000, B 0.000, C 0.000 }
gfCNCPoint4[7942] = {X 274.6929, Y 63.0558, Z -5.5000, A 0.000, B 0.000, C 0.000 }
gfCNCPoint4[7943] = {X 273.8964, Y 62.6626, Z -5.5000, A 0.000, B 0.000, C 0.000 }
gfCNCPoint4[7944] = {X 273.1952, Y 62.1174, Z -5.5000, A 0.000, B 0.000, C 0.000 }
gfCNCPoint4[7945] = {X 272.6178, Y 61.4425, Z -5.5000, A 0.000, B 0.000, C 0.000 }
gfCNCPoint4[7946] = {X 272.1876, Y 60.6654, Z -5.5000, A 0.000, B 0.000, C 0.000 }
gfCNCPoint4[7947] = {X 271.9223, Y 59.8177, Z -5.5000, A 0.000, B 0.000, C 0.000 }
gfCNCPoint4[7948] = {X 271.8327, Y 58.9341, Z -5.5000, A 0.000, B 0.000, C 0.000 }
gfCNCPoint4[7949] = {X 271.8327, Y 58.0000, Z -5.5000, A 0.000, B 0.000, C 0.000 }
gfCNCPoint4[7950] = {X 271.9430, Y 57.0209, Z -5.5000, A 0.000, B 0.000, C 0.000 }
gfCNCPoint4[7951] = {X 272.2684, Y 56.0909, Z -5.5000, A 0.000, B 0.000, C 0.000 }
gfCNCPoint4[7952] = {X 272.7926, Y 55.2566, Z -5.5000, A 0.000, B 0.000, C 0.000 }
gfCNCPoint4[7953] = {X 273.4893, Y 54.5599, Z -5.5000, A 0.000, B 0.000, C 0.000 }
gfCNCPoint4[7954] = {X 274.3236, Y 54.0357, Z -5.5000, A 0.000, B 0.000, C 0.000 }
gfCNCPoint4[7955] = {X 275.2536, Y 53.7103, Z -5.5000, A 0.000, B 0.000, C 0.000 }
gfCNCPoint4[7956] = {X 276.2327, Y 53.6000, Z -5.5000, A 0.000, B 0.000, C 0.000 }
gfCNCPoint4[7957] = {X 292.7731, Y 53.6000, Z -5.5000, A 0.000, B 0.000, C 0.000 }
gfCNCPoint4[7958] = {X 293.7522, Y 53.7103, Z -5.5000, A 0.000, B 0.000, C 0.000 }
gfCNCPoint4[7959] = {X 294.6822, Y 54.0357, Z -5.5000, A 0.000, B 0.000, C 0.000 }
gfCNCPoint4[7960] = {X 295.5164, Y 54.5599, Z -5.5000, A 0.000, B 0.000, C 0.000 }
gfCNCPoint4[7961] = {X 296.2131, Y 55.2566, Z -5.5000, A 0.000, B 0.000, C 0.000 }
gfCNCPoint4[7962] = {X 296.7373, Y 56.0909, Z -5.5000, A 0.000, B 0.000, C 0.000 }
gfCNCPoint4[7963] = {X 297.0628, Y 57.0209, Z -5.5000, A 0.000, B 0.000, C 0.000 }
gfCNCPoint4[7964] = {X 297.1731, Y 58.0000, Z -5.5000, A 0.000, B 0.000, C 0.000 }
gfCNCPoint4[7965] = {X 297.1731, Y 58.9353, Z -5.5000, A 0.000, B 0.000, C 0.000 }
gfCNCPoint4[7966] = {X 297.0812, Y 59.8183, Z -5.5000, A 0.000, B 0.000, C 0.000 }
gfCNCPoint4[7967] = {X 296.8146, Y 60.6650, Z -5.5000, A 0.000, B 0.000, C 0.000 }
gfCNCPoint4[7968] = {X 296.3840, Y 61.4414, Z -5.5000, A 0.000, B 0.000, C 0.000 }
gfCNCPoint4[7969] = {X 295.8069, Y 62.1159, Z -5.5000, A 0.000, B 0.000, C 0.000 }
gfCNCPoint4[7970] = {X 295.1065, Y 62.6614, Z -5.5000, A 0.000, B 0.000, C 0.000 }
gfCNCPoint4[7971] = {X 294.3112, Y 63.0558, Z -5.5000, A 0.000, B 0.000, C 0.000 }
gfCNCPoint4[7972] = {X 293.4531, Y 63.2832, Z -5.5000, A 0.000, B 0.000, C 0.000 }
gfCNCPoint4[7973] = {X 293.4531, Y 92.7105, Z -5.5000, A 0.000, B 0.000, C 0.000 }
gfCNCPoint4[7974] = {X 294.3110, Y 92.9404, Z -5.5000, A 0.000, B 0.000, C 0.000 }
gfCNCPoint4[7975] = {X 295.1058, Y 93.3367, Z -5.5000, A 0.000, B 0.000, C 0.000 }
gfCNCPoint4[7976] = {X 295.8057, Y 93.8835, Z -5.5000, A 0.000, B 0.000, C 0.000 }
gfCNCPoint4[7977] = {X 296.3825, Y 94.5589, Z -5.5000, A 0.000, B 0.000, C 0.000 }
gfCNCPoint4[7978] = {X 296.8131, Y 95.3357, Z -5.5000, A 0.000, B 0.000, C 0.000 }
gfCNCPoint4[7979] = {X 297.0802, Y 96.1828, Z -5.5000, A 0.000, B 0.000, C 0.000 }
gfCNCPoint4[7980] = {X 297.1731, Y 97.0661, Z -5.5000, A 0.000, B 0.000, C 0.000 }
gfCNCPoint4[7981] = {X 297.1731, Y 97.6951, Z -5.5000, A 0.000, B 0.000, C 0.000 }
gfCNCPoint4[7982] = {X 297.6531, Y 97.6951, Z -5.5000, A 0.000, B 0.000, C 0.000 }
gfCNCPoint4[7983] = {X 314.2122, Y 97.6951, Z -5.5000, A 0.000, B 0.000, C 0.000 }
gfCNCPoint4[7984] = {X 313.0149, Y 96.8448, Z -5.5000, A 0.000, B 0.000, C 0.000 }
gfCNCPoint4[7985] = {X 311.8816, Y 95.9109, Z -5.5000, A 0.000, B 0.000, C 0.000 }
gfCNCPoint4[7986] = {X 310.9059, Y 94.9488, Z -5.5000, A 0.000, B 0.000, C 0.000 }
gfCNCPoint4[7987] = {X 310.0415, Y 93.8856, Z -5.5000, A 0.000, B 0.000, C 0.000 }
gfCNCPoint4[7988] = {X 309.2075, Y 92.5709, Z -5.5000, A 0.000, B 0.000, C 0.000 }
gfCNCPoint4[7989] = {X 308.5436, Y 91.1626, Z -5.5000, A 0.000, B 0.000, C 0.000 }
gfCNCPoint4[7990] = {X 308.0602, Y 89.6827, Z -5.5000, A 0.000, B 0.000, C 0.000 }
gfCNCPoint4[7991] = {X 307.7067, Y 88.0128, Z -5.5000, A 0.000, B 0.000, C 0.000 }
gfCNCPoint4[7992] = {X 307.4978, Y 86.3188, Z -5.5000, A 0.000, B 0.000, C 0.000 }
gfCNCPoint4[7993] = {X 307.4350, Y 84.6131, Z -5.5000, A 0.000, B 0.000, C 0.000 }
gfCNCPoint4[7994] = {X 307.4363, Y 63.6742, Z -5.5000, A 0.000, B 0.000, C 0.000 }
gfCNCPoint4[7995] = {X 306.4279, Y 63.3059, Z -5.5000, A 0.000, B 0.000, C 0.000 }
gfCNCPoint4[7996] = {X 305.5245, Y 62.7260, Z -5.5000, A 0.000, B 0.000, C 0.000 }
gfCNCPoint4[7997] = {X 304.7698, Y 61.9627, Z -5.5000, A 0.000, B 0.000, C 0.000 }
gfCNCPoint4[7998] = {X 304.2001, Y 61.0528, Z -5.5000, A 0.000, B 0.000, C 0.000 }
gfCNCPoint4[7999] = {X 303.8433, Y 60.0403, Z -5.5000, A 0.000, B 0.000, C 0.000 }
gfCNCPoint4[8000] = {X 303.7164, Y 58.9744, Z -5.5000, A 0.000, B 0.000, C 0.000 }
gfCNCPoint4[8001] = {X 303.7162, Y 58.0000, Z -5.5000, A 0.000, B 0.000, C 0.000 }
gfCNCPoint4[8002] = {X 303.8100, Y 57.0480, Z -5.5000, A 0.000, B 0.000, C 0.000 }
gfCNCPoint4[8003] = {X 304.0877, Y 56.1325, Z -5.5000, A 0.000, B 0.000, C 0.000 }
gfCNCPoint4[8004] = {X 304.5387, Y 55.2888, Z -5.5000, A 0.000, B 0.000, C 0.000 }
gfCNCPoint4[8005] = {X 305.1455, Y 54.5493, Z -5.5000, A 0.000, B 0.000, C 0.000 }
gfCNCPoint4[8006] = {X 305.8850, Y 53.9424, Z -5.5000, A 0.000, B 0.000, C 0.000 }
gfCNCPoint4[8007] = {X 306.7287, Y 53.4915, Z -5.5000, A 0.000, B 0.000, C 0.000 }
gfCNCPoint4[8008] = {X 307.6442, Y 53.2138, Z -5.5000, A 0.000, B 0.000, C 0.000 }
gfCNCPoint4[8009] = {X 308.5962, Y 53.1200, Z -5.5000, A 0.000, B 0.000, C 0.000 }
gfCNCPoint4[8010] = {X 324.3107, Y 53.1200, Z -5.5000, A 0.000, B 0.000, C 0.000 }
gfCNCPoint4[8011] = {X 325.2627, Y 53.2138, Z -5.5000, A 0.000, B 0.000, C 0.000 }
gfCNCPoint4[8012] = {X 326.1782, Y 53.4915, Z -5.5000, A 0.000, B 0.000, C 0.000 }
gfCNCPoint4[8013] = {X 327.0219, Y 53.9424, Z -5.5000, A 0.000, B 0.000, C 0.000 }
gfCNCPoint4[8014] = {X 327.7614, Y 54.5493, Z -5.5000, A 0.000, B 0.000, C 0.000 }
gfCNCPoint4[8015] = {X 328.3683, Y 55.2888, Z -5.5000, A 0.000, B 0.000, C 0.000 }
gfCNCPoint4[8016] = {X 328.8192, Y 56.1325, Z -5.5000, A 0.000, B 0.000, C 0.000 }
gfCNCPoint4[8017] = {X 329.0969, Y 57.0480, Z -5.5000, A 0.000, B 0.000, C 0.000 }
gfCNCPoint4[8018] = {X 329.1907, Y 58.0000, Z -5.5000, A 0.000, B 0.000, C 0.000 }
gfCNCPoint4[8019] = {X 329.1907, Y 58.9341, Z -5.5000, A 0.000, B 0.000, C 0.000 }
gfCNCPoint4[8020] = {X 329.0673, Y 60.0067, Z -5.5000, A 0.000, B 0.000, C 0.000 }
gfCNCPoint4[8021] = {X 328.7127, Y 61.0266, Z -5.5000, A 0.000, B 0.000, C 0.000 }
gfCNCPoint4[8022] = {X 328.1442, Y 61.9445, Z -5.5000, A 0.000, B 0.000, C 0.000 }
gfCNCPoint4[8023] = {X 327.3891, Y 62.7163, Z -5.5000, A 0.000, B 0.000, C 0.000 }
gfCNCPoint4[8024] = {X 326.4838, Y 63.3046, Z -5.5000, A 0.000, B 0.000, C 0.000 }
gfCNCPoint4[8025] = {X 325.4719, Y 63.6812, Z -5.5000, A 0.000, B 0.000, C 0.000 }
gfCNCPoint4[8026] = {X 325.4736, Y 83.2269, Z -5.5000, A 0.000, B 0.000, C 0.000 }
gfCNCPoint4[8027] = {X 325.4871, Y 84.6073, Z -5.5000, A 0.000, B 0.000, C 0.000 }
gfCNCPoint4[8028] = {X 325.5530, Y 85.7200, Z -5.5000, A 0.000, B 0.000, C 0.000 }
gfCNCPoint4[8029] = {X 325.7426, Y 86.8183, Z -5.5000, A 0.000, B 0.000, C 0.000 }
gfCNCPoint4[8030] = {X 325.8867, Y 86.9524, Z -5.5000, A 0.000, B 0.000, C 0.000 }
gfCNCPoint4[8031] = {X 326.0551, Y 87.0543, Z -5.5000, A 0.000, B 0.000, C 0.000 }
gfCNCPoint4[8032] = {X 326.4842, Y 87.2970, Z -5.5000, A 0.000, B 0.000, C 0.000 }
gfCNCPoint4[8033] = {X 327.8572, Y 87.8650, Z -5.5000, A 0.000, B 0.000, C 0.000 }
gfCNCPoint4[8034] = {X 329.2839, Y 88.2803, Z -5.5000, A 0.000, B 0.000, C 0.000 }
gfCNCPoint4[8035] = {X 331.5313, Y 88.7482, Z -5.5000, A 0.000, B 0.000, C 0.000 }
gfCNCPoint4[8036] = {X 333.7991, Y 89.1051, Z -5.5000, A 0.000, B 0.000, C 0.000 }
gfCNCPoint4[8037] = {X 336.0816, Y 89.3502, Z -5.5000, A 0.000, B 0.000, C 0.000 }
gfCNCPoint4[8038] = {X 340.4337, Y 89.6433, Z -5.5000, A 0.000, B 0.000, C 0.000 }
gfCNCPoint4[8039] = {X 344.7930, Y 89.7965, Z -5.5000, A 0.000, B 0.000, C 0.000 }
gfCNCPoint4[8040] = {X 349.1549, Y 89.8097, Z -5.5000, A 0.000, B 0.000, C 0.000 }
gfCNCPoint4[8041] = {X 353.2889, Y 89.7420, Z -5.5000, A 0.000, B 0.000, C 0.000 }
gfCNCPoint4[8042] = {X 357.4177, Y 89.5240, Z -5.5000, A 0.000, B 0.000, C 0.000 }
gfCNCPoint4[8043] = {X 361.5359, Y 89.1563, Z -5.5000, A 0.000, B 0.000, C 0.000 }
gfCNCPoint4[8044] = {X 363.5861, Y 88.8735, Z -5.5000, A 0.000, B 0.000, C 0.000 }
gfCNCPoint4[8045] = {X 365.6175, Y 88.4774, Z -5.5000, A 0.000, B 0.000, C 0.000 }
gfCNCPoint4[8046] = {X 367.6239, Y 87.9694, Z -5.5000, A 0.000, B 0.000, C 0.000 }
gfCNCPoint4[8047] = {X 368.9177, Y 87.4946, Z -5.5000, A 0.000, B 0.000, C 0.000 }
gfCNCPoint4[8048] = {X 370.1137, Y 86.8096, Z -5.5000, A 0.000, B 0.000, C 0.000 }
gfCNCPoint4[8049] = {X 370.2982, Y 85.3241, Z -5.5000, A 0.000, B 0.000, C 0.000 }
gfCNCPoint4[8050] = {X 370.3597, Y 83.8285, Z -5.5000, A 0.000, B 0.000, C 0.000 }
gfCNCPoint4[8051] = {X 370.3584, Y 63.6740, Z -5.5000, A 0.000, B 0.000, C 0.000 }
gfCNCPoint4[8052] = {X 369.3503, Y 63.3055, Z -5.5000, A 0.000, B 0.000, C 0.000 }
gfCNCPoint4[8053] = {X 368.4471, Y 62.7256, Z -5.5000, A 0.000, B 0.000, C 0.000 }
gfCNCPoint4[8054] = {X 367.6925, Y 61.9623, Z -5.5000, A 0.000, B 0.000, C 0.000 }
gfCNCPoint4[8055] = {X 367.1231, Y 61.0525, Z -5.5000, A 0.000, B 0.000, C 0.000 }
gfCNCPoint4[8056] = {X 366.7663, Y 60.0402, Z -5.5000, A 0.000, B 0.000, C 0.000 }
gfCNCPoint4[8057] = {X 366.6394, Y 58.9744, Z -5.5000, A 0.000, B 0.000, C 0.000 }
gfCNCPoint4[8058] = {X 366.6393, Y 58.0000, Z -5.5000, A 0.000, B 0.000, C 0.000 }
gfCNCPoint4[8059] = {X 366.7331, Y 57.0480, Z -5.5000, A 0.000, B 0.000, C 0.000 }
gfCNCPoint4[8060] = {X 367.0108, Y 56.1325, Z -5.5000, A 0.000, B 0.000, C 0.000 }
gfCNCPoint4[8061] = {X 367.4617, Y 55.2888, Z -5.5000, A 0.000, B 0.000, C 0.000 }
gfCNCPoint4[8062] = {X 368.0686, Y 54.5493, Z -5.5000, A 0.000, B 0.000, C 0.000 }
gfCNCPoint4[8063] = {X 368.8081, Y 53.9424, Z -5.5000, A 0.000, B 0.000, C 0.000 }
gfCNCPoint4[8064] = {X 369.6518, Y 53.4915, Z -5.5000, A 0.000, B 0.000, C 0.000 }
gfCNCPoint4[8065] = {X 370.5672, Y 53.2138, Z -5.5000, A 0.000, B 0.000, C 0.000 }
gfCNCPoint4[8066] = {X 371.5193, Y 53.1200, Z -5.5000, A 0.000, B 0.000, C 0.000 }
gfCNCPoint4[8067] = {X 388.0597, Y 53.1200, Z -5.5000, A 0.000, B 0.000, C 0.000 }
gfCNCPoint4[8068] = {X 389.0355, Y 53.2186, Z -5.5000, A 0.000, B 0.000, C 0.000 }
gfCNCPoint4[8069] = {X 389.9719, Y 53.5102, Z -5.5000, A 0.000, B 0.000, C 0.000 }
gfCNCPoint4[8070] = {X 390.8310, Y 53.9833, Z -5.5000, A 0.000, B 0.000, C 0.000 }
gfCNCPoint4[8071] = {X 391.5783, Y 54.6186, Z -5.5000, A 0.000, B 0.000, C 0.000 }
gfCNCPoint4[8072] = {X 392.1572, Y 55.3496, Z -5.5000, A 0.000, B 0.000, C 0.000 }
gfCNCPoint4[8073] = {X 392.5865, Y 56.1774, Z -5.5000, A 0.000, B 0.000, C 0.000 }
gfCNCPoint4[8074] = {X 392.8506, Y 57.0718, Z -5.5000, A 0.000, B 0.000, C 0.000 }
gfCNCPoint4[8075] = {X 392.9397, Y 58.0000, Z -5.5000, A 0.000, B 0.000, C 0.000 }
gfCNCPoint4[8076] = {X 392.9395, Y 58.9744, Z -5.5000, A 0.000, B 0.000, C 0.000 }
gfCNCPoint4[8077] = {X 392.8786, Y 59.7035, Z -5.5000, A 0.000, B 0.000, C 0.000 }
gfCNCPoint4[8078] = {X 392.7094, Y 60.4153, Z -5.5000, A 0.000, B 0.000, C 0.000 }
gfCNCPoint4[8079] = {X 392.4357, Y 61.0938, Z -5.5000, A 0.000, B 0.000, C 0.000 }
gfCNCPoint4[8080] = {X 392.0535, Y 61.7388, Z -5.5000, A 0.000, B 0.000, C 0.000 }
gfCNCPoint4[8081] = {X 391.5774, Y 62.3179, Z -5.5000, A 0.000, B 0.000, C 0.000 }
gfCNCPoint4[8082] = {X 390.8819, Y 62.9185, Z -5.5000, A 0.000, B 0.000, C 0.000 }
gfCNCPoint4[8083] = {X 390.0866, Y 63.3788, Z -5.5000, A 0.000, B 0.000, C 0.000 }
gfCNCPoint4[8084] = {X 389.2193, Y 63.6826, Z -5.5000, A 0.000, B 0.000, C 0.000 }
gfCNCPoint4[8085] = {X 389.2184, Y 73.4819, Z -5.5000, A 0.000, B 0.000, C 0.000 }
gfCNCPoint4[8086] = {X 398.8184, Y 73.4828, Z -5.5000, A 0.000, B 0.000, C 0.000 }
gfCNCPoint4[8087] = {X 398.8177, Y 80.5573, Z -5.5000, A 0.000, B 0.000, C 0.000 }
gfCNCPoint4[8088] = {X 405.8031, Y 76.0835, Z -5.5000, A 0.000, B 0.000, C 0.000 }
gfCNCPoint4[8089] = {X 400.0380, Y 73.8217, Z -5.5000, A 0.000, B 0.000, C 0.000 }
gfCNCPoint4[8090] = {X 399.4370, Y 73.6206, Z -5.5000, A 0.000, B 0.000, C 0.000 }
gfCNCPoint4[8091] = {X 398.8184, Y 73.4828, Z -5.5000, A 0.000, B 0.000, C 0.000 }
gfCNCPoint4[8092] = {X 396.4184, Y 73.4826, Z -5.5000, A 0.000, B 0.000, C 0.000 }
gfCNCPoint4[8093] = {X 396.4173, Y 84.5897, Z -5.5000, A 0.000, B 0.000, C 0.000 }
gfCNCPoint4[8094] = {X 396.4172, Y 84.9446, Z -5.5000, A 0.000, B 0.000, C 0.000 }
gfCNCPoint4[8095] = {X 411.0590, Y 75.5675, Z -5.5000, A 0.000, B 0.000, C 0.000 }
gfCNCPoint4[8096] = {X 400.9163, Y 71.5881, Z -5.5000, A 0.000, B 0.000, C 0.000 }
gfCNCPoint4[8097] = {X 399.6200, Y 71.1942, Z -5.5000, A 0.000, B 0.000, C 0.000 }
gfCNCPoint4[8098] = {X 398.2776, Y 71.0108, Z -5.5000, A 0.000, B 0.000, C 0.000 }
gfCNCPoint4[8099] = {X 397.3445, Y 70.9530, Z -5.5000, A 0.000, B 0.000, C 0.000 }
gfCNCPoint4[8100] = {X 396.4186, Y 70.8232, Z -5.5000, A 0.000, B 0.000, C 0.000 }
gfCNCPoint4[8101] = {X 396.4184, Y 73.4826, Z -5.5000, A 0.000, B 0.000, C 0.000 }
gfCNCPoint4[8102] = {X 394.0184, Y 73.4824, Z -5.5000, A 0.000, B 0.000, C 0.000 }
gfCNCPoint4[8103] = {X 394.0173, Y 84.5973, Z -5.5000, A 0.000, B 0.000, C 0.000 }
gfCNCPoint4[8104] = {X 394.0178, Y 84.7626, Z -5.5000, A 0.000, B 0.000, C 0.000 }
gfCNCPoint4[8105] = {X 394.0172, Y 84.9279, Z -5.5000, A 0.000, B 0.000, C 0.000 }
gfCNCPoint4[8106] = {X 393.9669, Y 86.3333, Z -5.5000, A 0.000, B 0.000, C 0.000 }
gfCNCPoint4[8107] = {X 393.8355, Y 87.7335, Z -5.5000, A 0.000, B 0.000, C 0.000 }
gfCNCPoint4[8108] = {X 395.0834, Y 87.4767, Z -5.5000, A 0.000, B 0.000, C 0.000 }
gfCNCPoint4[8109] = {X 396.3542, Y 87.3861, Z -5.5000, A 0.000, B 0.000, C 0.000 }
gfCNCPoint4[8110] = {X 396.7363, Y 87.3713, Z -5.5000, A 0.000, B 0.000, C 0.000 }
gfCNCPoint4[8111] = {X 397.1179, Y 87.3459, Z -5.5000, A 0.000, B 0.000, C 0.000 }
gfCNCPoint4[8112] = {X 416.3148, Y 75.0515, Z -5.5000, A 0.000, B 0.000, C 0.000 }
gfCNCPoint4[8113] = {X 401.7945, Y 69.3546, Z -5.5000, A 0.000, B 0.000, C 0.000 }
gfCNCPoint4[8114] = {X 400.6812, Y 68.9846, Z -5.5000, A 0.000, B 0.000, C 0.000 }
gfCNCPoint4[8115] = {X 399.5347, Y 68.7362, Z -5.5000, A 0.000, B 0.000, C 0.000 }
gfCNCPoint4[8116] = {X 398.3682, Y 68.6122, Z -5.5000, A 0.000, B 0.000, C 0.000 }
gfCNCPoint4[8117] = {X 397.6029, Y 68.5669, Z -5.5000, A 0.000, B 0.000, C 0.000 }
gfCNCPoint4[8118] = {X 396.8436, Y 68.4611, Z -5.5000, A 0.000, B 0.000, C 0.000 }
gfCNCPoint4[8119] = {X 395.3933, Y 68.0822, Z -5.5000, A 0.000, B 0.000, C 0.000 }
gfCNCPoint4[8120] = {X 394.0189, Y 67.4840, Z -5.5000, A 0.000, B 0.000, C 0.000 }
gfCNCPoint4[8121] = {X 394.0184, Y 73.4824, Z -5.5000, A 0.000, B 0.000, C 0.000 }
gfCNCPoint4[8122] = {X 391.6184, Y 73.4821, Z -5.5000, A 0.000, B 0.000, C 0.000 }
gfCNCPoint4[8123] = {X 391.6173, Y 84.6054, Z -5.5000, A 0.000, B 0.000, C 0.000 }
gfCNCPoint4[8124] = {X 391.5812, Y 86.0255, Z -5.5000, A 0.000, B 0.000, C 0.000 }
gfCNCPoint4[8125] = {X 391.4535, Y 87.4404, Z -5.5000, A 0.000, B 0.000, C 0.000 }
gfCNCPoint4[8126] = {X 391.2291, Y 88.8723, Z -5.5000, A 0.000, B 0.000, C 0.000 }
gfCNCPoint4[8127] = {X 390.9109, Y 90.2862, Z -5.5000, A 0.000, B 0.000, C 0.000 }
gfCNCPoint4[8128] = {X 390.3346, Y 92.0501, Z -5.5000, A 0.000, B 0.000, C 0.000 }
gfCNCPoint4[8129] = {X 389.5432, Y 93.7284, Z -5.5000, A 0.000, B 0.000, C 0.000 }
gfCNCPoint4[8130] = {X 388.5488, Y 95.2951, Z -5.5000, A 0.000, B 0.000, C 0.000 }
gfCNCPoint4[8131] = {X 389.3446, Y 95.2951, Z -5.5000, A 0.000, B 0.000, C 0.000 }
gfCNCPoint4[8132] = {X 389.7639, Y 94.0857, Z -5.5000, A 0.000, B 0.000, C 0.000 }
gfCNCPoint4[8133] = {X 390.3886, Y 92.9684, Z -5.5000, A 0.000, B 0.000, C 0.000 }
gfCNCPoint4[8134] = {X 391.1992, Y 91.9779, Z -5.5000, A 0.000, B 0.000, C 0.000 }
gfCNCPoint4[8135] = {X 392.1709, Y 91.1446, Z -5.5000, A 0.000, B 0.000, C 0.000 }
gfCNCPoint4[8136] = {X 393.2734, Y 90.4944, Z -5.5000, A 0.000, B 0.000, C 0.000 }
gfCNCPoint4[8137] = {X 394.4728, Y 90.0473, Z -5.5000, A 0.000, B 0.000, C 0.000 }
gfCNCPoint4[8138] = {X 395.4216, Y 89.8528, Z -5.5000, A 0.000, B 0.000, C 0.000 }
gfCNCPoint4[8139] = {X 396.3879, Y 89.7860, Z -5.5000, A 0.000, B 0.000, C 0.000 }
gfCNCPoint4[8140] = {X 397.1572, Y 89.7497, Z -5.5000, A 0.000, B 0.000, C 0.000 }
gfCNCPoint4[8141] = {X 397.9239, Y 89.6771, Z -5.5000, A 0.000, B 0.000, C 0.000 }
gfCNCPoint4[8142] = {X 417.6092, Y 77.0726, Z -5.5000, A 0.000, B 0.000, C 0.000 }
gfCNCPoint4[8143] = {X 421.5707, Y 74.5355, Z -5.5000, A 0.000, B 0.000, C 0.000 }
gfCNCPoint4[8144] = {X 402.6727, Y 67.1210, Z -5.5000, A 0.000, B 0.000, C 0.000 }
gfCNCPoint4[8145] = {X 401.3007, Y 66.6658, Z -5.5000, A 0.000, B 0.000, C 0.000 }
gfCNCPoint4[8146] = {X 399.8874, Y 66.3621, Z -5.5000, A 0.000, B 0.000, C 0.000 }
gfCNCPoint4[8147] = {X 398.4495, Y 66.2133, Z -5.5000, A 0.000, B 0.000, C 0.000 }
gfCNCPoint4[8148] = {X 397.3052, Y 66.1055, Z -5.5000, A 0.000, B 0.000, C 0.000 }
gfCNCPoint4[8149] = {X 396.1920, Y 65.8190, Z -5.5000, A 0.000, B 0.000, C 0.000 }
gfCNCPoint4[8150] = {X 395.1378, Y 65.3608, Z -5.5000, A 0.000, B 0.000, C 0.000 }
gfCNCPoint4[8151] = {X 394.1689, Y 64.7424, Z -5.5000, A 0.000, B 0.000, C 0.000 }
gfCNCPoint4[8152] = {X 393.3094, Y 63.9792, Z -5.5000, A 0.000, B 0.000, C 0.000 }
gfCNCPoint4[8153] = {X 392.5125, Y 64.6964, Z -5.5000, A 0.000, B 0.000, C 0.000 }
gfCNCPoint4[8154] = {X 391.6191, Y 65.2891, Z -5.5000, A 0.000, B 0.000, C 0.000 }
gfCNCPoint4[8155] = {X 391.6184, Y 73.4821, Z -5.5000, A 0.000, B 0.000, C 0.000 }
gfCNCPoint4[8156] = {X 389.2184, Y 73.4819, Z -5.5000, A 0.000, B 0.000, C 0.000 }
gfCNCPoint4[8157] = {X 389.2173, Y 84.6139, Z -5.5000, A 0.000, B 0.000, C 0.000 }
gfCNCPoint4[8158] = {X 389.1554, Y 86.3199, Z -5.5000, A 0.000, B 0.000, C 0.000 }
gfCNCPoint4[8159] = {X 388.9450, Y 88.0141, Z -5.5000, A 0.000, B 0.000, C 0.000 }
gfCNCPoint4[8160] = {X 388.5878, Y 89.6835, Z -5.5000, A 0.000, B 0.000, C 0.000 }
gfCNCPoint4[8161] = {X 388.1046, Y 91.1631, Z -5.5000, A 0.000, B 0.000, C 0.000 }
gfCNCPoint4[8162] = {X 387.4408, Y 92.5709, Z -5.5000, A 0.000, B 0.000, C 0.000 }
gfCNCPoint4[8163] = {X 386.6067, Y 93.8850, Z -5.5000, A 0.000, B 0.000, C 0.000 }
gfCNCPoint4[8164] = {X 385.8746, Y 94.7997, Z -5.5000, A 0.000, B 0.000, C 0.000 }
gfCNCPoint4[8165] = {X 385.0599, Y 95.6417, Z -5.5000, A 0.000, B 0.000, C 0.000 }
gfCNCPoint4[8166] = {X 383.8000, Y 96.7249, Z -5.5000, A 0.000, B 0.000, C 0.000 }
gfCNCPoint4[8167] = {X 382.4511, Y 97.6951, Z -5.5000, A 0.000, B 0.000, C 0.000 }
gfCNCPoint4[8168] = {X 382.1880, Y 97.2936, Z -5.5000, A 0.000, B 0.000, C 0.000 }
gfCNCPoint4[8169] = {X 381.0201, Y 97.9996, Z -5.5000, A 0.000, B 0.000, C 0.000 }
gfCNCPoint4[8170] = {X 379.8040, Y 98.6185, Z -5.5000, A 0.000, B 0.000, C 0.000 }
gfCNCPoint4[8171] = {X 377.5267, Y 99.5759, Z -5.5000, A 0.000, B 0.000, C 0.000 }
gfCNCPoint4[8172] = {X 375.1867, Y 100.3681, Z -5.5000, A 0.000, B 0.000, C 0.000 }
gfCNCPoint4[8173] = {X 372.7962, Y 100.9910, Z -5.5000, A 0.000, B 0.000, C 0.000 }
gfCNCPoint4[8174] = {X 368.8821, Y 101.7457, Z -5.5000, A 0.000, B 0.000, C 0.000 }
gfCNCPoint4[8175] = {X 364.9355, Y 102.3065, Z -5.5000, A 0.000, B 0.000, C 0.000 }
gfCNCPoint4[8176] = {X 360.9660, Y 102.6719, Z -5.5000, A 0.000, B 0.000, C 0.000 }
gfCNCPoint4[8177] = {X 355.2456, Y 102.9770, Z -5.5000, A 0.000, B 0.000, C 0.000 }
gfCNCPoint4[8178] = {X 349.5186, Y 103.1071, Z -5.5000, A 0.000, B 0.000, C 0.000 }
gfCNCPoint4[8179] = {X 343.7903, Y 103.0621, Z -5.5000, A 0.000, B 0.000, C 0.000 }
gfCNCPoint4[8180] = {X 338.0660, Y 102.8420, Z -5.5000, A 0.000, B 0.000, C 0.000 }
gfCNCPoint4[8181] = {X 334.1085, Y 102.5649, Z -5.5000, A 0.000, B 0.000, C 0.000 }
gfCNCPoint4[8182] = {X 330.1660, Y 102.1227, Z -5.5000, A 0.000, B 0.000, C 0.000 }
gfCNCPoint4[8183] = {X 326.2454, Y 101.5162, Z -5.5000, A 0.000, B 0.000, C 0.000 }
gfCNCPoint4[8184] = {X 323.3899, Y 100.9106, Z -5.5000, A 0.000, B 0.000, C 0.000 }
gfCNCPoint4[8185] = {X 320.5870, Y 100.0961, Z -5.5000, A 0.000, B 0.000, C 0.000 }
gfCNCPoint4[8186] = {X 317.8518, Y 99.0769, Z -5.5000, A 0.000, B 0.000, C 0.000 }
gfCNCPoint4[8187] = {X 316.3328, Y 98.3765, Z -5.5000, A 0.000, B 0.000, C 0.000 }
gfCNCPoint4[8188] = {X 314.8777, Y 97.5514, Z -5.5000, A 0.000, B 0.000, C 0.000 }
gfCNCPoint4[8189] = {X 313.4968, Y 96.6075, Z -5.5000, A 0.000, B 0.000, C 0.000 }
gfCNCPoint4[8190] = {X 312.1997, Y 95.5514, Z -5.5000, A 0.000, B 0.000, C 0.000 }
gfCNCPoint4[8191] = {X 311.1891, Y 94.5460, Z -5.5000, A 0.000, B 0.000, C 0.000 }
gfCNCPoint4[8192] = {X 310.3048, Y 93.4279, Z -5.5000, A 0.000, B 0.000, C 0.000 }
gfCNCPoint4[8193] = {X 309.5594, Y 92.2129, Z -5.5000, A 0.000, B 0.000, C 0.000 }
gfCNCPoint4[8194] = {X 308.9632, Y 90.9180, Z -5.5000, A 0.000, B 0.000, C 0.000 }
gfCNCPoint4[8195] = {X 308.5247, Y 89.5616, Z -5.5000, A 0.000, B 0.000, C 0.000 }
gfCNCPoint4[8196] = {X 308.1799, Y 87.9321, Z -5.5000, A 0.000, B 0.000, C 0.000 }
gfCNCPoint4[8197] = {X 307.9762, Y 86.2791, Z -5.5000, A 0.000, B 0.000, C 0.000 }
gfCNCPoint4[8198] = {X 307.9150, Y 84.6146, Z -5.5000, A 0.000, B 0.000, C 0.000 }
gfCNCPoint4[8199] = {X 307.9163, Y 63.2812, Z -5.5000, A 0.000, B 0.000, C 0.000 }
gfCNCPoint4[8200] = {X 307.0570, Y 63.0560, Z -5.5000, A 0.000, B 0.000, C 0.000 }
gfCNCPoint4[8201] = {X 306.2604, Y 62.6629, Z -5.5000, A 0.000, B 0.000, C 0.000 }
gfCNCPoint4[8202] = {X 305.5591, Y 62.1177, Z -5.5000, A 0.000, B 0.000, C 0.000 }
gfCNCPoint4[8203] = {X 304.9815, Y 61.4428, Z -5.5000, A 0.000, B 0.000, C 0.000 }
gfCNCPoint4[8204] = {X 304.5513, Y 60.6656, Z -5.5000, A 0.000, B 0.000, C 0.000 }
gfCNCPoint4[8205] = {X 304.2859, Y 59.8178, Z -5.5000, A 0.000, B 0.000, C 0.000 }
gfCNCPoint4[8206] = {X 304.1962, Y 58.9341, Z -5.5000, A 0.000, B 0.000, C 0.000 }
gfCNCPoint4[8207] = {X 304.1962, Y 58.0000, Z -5.5000, A 0.000, B 0.000, C 0.000 }
gfCNCPoint4[8208] = {X 304.3065, Y 57.0209, Z -5.5000, A 0.000, B 0.000, C 0.000 }
gfCNCPoint4[8209] = {X 304.6320, Y 56.0909, Z -5.5000, A 0.000, B 0.000, C 0.000 }
gfCNCPoint4[8210] = {X 305.1562, Y 55.2566, Z -5.5000, A 0.000, B 0.000, C 0.000 }
gfCNCPoint4[8211] = {X 305.8529, Y 54.5599, Z -5.5000, A 0.000, B 0.000, C 0.000 }
gfCNCPoint4[8212] = {X 306.6871, Y 54.0357, Z -5.5000, A 0.000, B 0.000, C 0.000 }
gfCNCPoint4[8213] = {X 307.6171, Y 53.7103, Z -5.5000, A 0.000, B 0.000, C 0.000 }
gfCNCPoint4[8214] = {X 308.5962, Y 53.6000, Z -5.5000, A 0.000, B 0.000, C 0.000 }
gfCNCPoint4[8215] = {X 324.3107, Y 53.6000, Z -5.5000, A 0.000, B 0.000, C 0.000 }
gfCNCPoint4[8216] = {X 325.2898, Y 53.7103, Z -5.5000, A 0.000, B 0.000, C 0.000 }
gfCNCPoint4[8217] = {X 326.2198, Y 54.0357, Z -5.5000, A 0.000, B 0.000, C 0.000 }
gfCNCPoint4[8218] = {X 327.0540, Y 54.5599, Z -5.5000, A 0.000, B 0.000, C 0.000 }
gfCNCPoint4[8219] = {X 327.7507, Y 55.2566, Z -5.5000, A 0.000, B 0.000, C 0.000 }
gfCNCPoint4[8220] = {X 328.2750, Y 56.0909, Z -5.5000, A 0.000, B 0.000, C 0.000 }
gfCNCPoint4[8221] = {X 328.6004, Y 57.0209, Z -5.5000, A 0.000, B 0.000, C 0.000 }
gfCNCPoint4[8222] = {X 328.7107, Y 58.0000, Z -5.5000, A 0.000, B 0.000, C 0.000 }
gfCNCPoint4[8223] = {X 328.7107, Y 58.9363, Z -5.5000, A 0.000, B 0.000, C 0.000 }
gfCNCPoint4[8224] = {X 328.6170, Y 59.8191, Z -5.5000, A 0.000, B 0.000, C 0.000 }
gfCNCPoint4[8225] = {X 328.3495, Y 60.6655, Z -5.5000, A 0.000, B 0.000, C 0.000 }
gfCNCPoint4[8226] = {X 327.9189, Y 61.4418, Z -5.5000, A 0.000, B 0.000, C 0.000 }
gfCNCPoint4[8227] = {X 327.3424, Y 62.1168, Z -5.5000, A 0.000, B 0.000, C 0.000 }
gfCNCPoint4[8228] = {X 326.6431, Y 62.6636, Z -5.5000, A 0.000, B 0.000, C 0.000 }
gfCNCPoint4[8229] = {X 325.8490, Y 63.0603, Z -5.5000, A 0.000, B 0.000, C 0.000 }
gfCNCPoint4[8230] = {X 324.9918, Y 63.2910, Z -5.5000, A 0.000, B 0.000, C 0.000 }
gfCNCPoint4[8231] = {X 324.9936, Y 83.2293, Z -5.5000, A 0.000, B 0.000, C 0.000 }
gfCNCPoint4[8232] = {X 325.0071, Y 84.6143, Z -5.5000, A 0.000, B 0.000, C 0.000 }
gfCNCPoint4[8233] = {X 325.0830, Y 85.8323, Z -5.5000, A 0.000, B 0.000, C 0.000 }
gfCNCPoint4[8234] = {X 325.3002, Y 87.0332, Z -5.5000, A 0.000, B 0.000, C 0.000 }
gfCNCPoint4[8235] = {X 325.5333, Y 87.2836, Z -5.5000, A 0.000, B 0.000, C 0.000 }
gfCNCPoint4[8236] = {X 325.8188, Y 87.4721, Z -5.5000, A 0.000, B 0.000, C 0.000 }
gfCNCPoint4[8237] = {X 326.2620, Y 87.7228, Z -5.5000, A 0.000, B 0.000, C 0.000 }
gfCNCPoint4[8238] = {X 327.6906, Y 88.3152, Z -5.5000, A 0.000, B 0.000, C 0.000 }
gfCNCPoint4[8239] = {X 329.1754, Y 88.7479, Z -5.5000, A 0.000, B 0.000, C 0.000 }
gfCNCPoint4[8240] = {X 331.4458, Y 89.2205, Z -5.5000, A 0.000, B 0.000, C 0.000 }
gfCNCPoint4[8241] = {X 333.7367, Y 89.5810, Z -5.5000, A 0.000, B 0.000, C 0.000 }
gfCNCPoint4[8242] = {X 336.0424, Y 89.8286, Z -5.5000, A 0.000, B 0.000, C 0.000 }
gfCNCPoint4[8243] = {X 340.4116, Y 90.1228, Z -5.5000, A 0.000, B 0.000, C 0.000 }
gfCNCPoint4[8244] = {X 344.7880, Y 90.2765, Z -5.5000, A 0.000, B 0.000, C 0.000 }
gfCNCPoint4[8245] = {X 349.1670, Y 90.2896, Z -5.5000, A 0.000, B 0.000, C 0.000 }
gfCNCPoint4[8246] = {X 353.3143, Y 90.2213, Z -5.5000, A 0.000, B 0.000, C 0.000 }
gfCNCPoint4[8247] = {X 357.4564, Y 90.0025, Z -5.5000, A 0.000, B 0.000, C 0.000 }
gfCNCPoint4[8248] = {X 361.5878, Y 89.6335, Z -5.5000, A 0.000, B 0.000, C 0.000 }
gfCNCPoint4[8249] = {X 363.6655, Y 89.3468, Z -5.5000, A 0.000, B 0.000, C 0.000 }
gfCNCPoint4[8250] = {X 365.7242, Y 88.9454, Z -5.5000, A 0.000, B 0.000, C 0.000 }
gfCNCPoint4[8251] = {X 367.7574, Y 88.4305, Z -5.5000, A 0.000, B 0.000, C 0.000 }
gfCNCPoint4[8252] = {X 368.6801, Y 88.1202, Z -5.5000, A 0.000, B 0.000, C 0.000 }
gfCNCPoint4[8253] = {X 369.5621, Y 87.7084, Z -5.5000, A 0.000, B 0.000, C 0.000 }
gfCNCPoint4[8254] = {X 370.3925, Y 87.2004, Z -5.5000, A 0.000, B 0.000, C 0.000 }
gfCNCPoint4[8255] = {X 370.5202, Y 87.0675, Z -5.5000, A 0.000, B 0.000, C 0.000 }
gfCNCPoint4[8256] = {X 370.5860, Y 86.8955, Z -5.5000, A 0.000, B 0.000, C 0.000 }
gfCNCPoint4[8257] = {X 370.7762, Y 85.3672, Z -5.5000, A 0.000, B 0.000, C 0.000 }
gfCNCPoint4[8258] = {X 370.8397, Y 83.8285, Z -5.5000, A 0.000, B 0.000, C 0.000 }
gfCNCPoint4[8259] = {X 370.8384, Y 63.2811, Z -5.5000, A 0.000, B 0.000, C 0.000 }
gfCNCPoint4[8260] = {X 369.9793, Y 63.0558, Z -5.5000, A 0.000, B 0.000, C 0.000 }
gfCNCPoint4[8261] = {X 369.1829, Y 62.6625, Z -5.5000, A 0.000, B 0.000, C 0.000 }
gfCNCPoint4[8262] = {X 368.4817, Y 62.1173, Z -5.5000, A 0.000, B 0.000, C 0.000 }
gfCNCPoint4[8263] = {X 367.9043, Y 61.4424, Z -5.5000, A 0.000, B 0.000, C 0.000 }
gfCNCPoint4[8264] = {X 367.4742, Y 60.6653, Z -5.5000, A 0.000, B 0.000, C 0.000 }
gfCNCPoint4[8265] = {X 367.2089, Y 59.8177, Z -5.5000, A 0.000, B 0.000, C 0.000 }
gfCNCPoint4[8266] = {X 367.1193, Y 58.9341, Z -5.5000, A 0.000, B 0.000, C 0.000 }
gfCNCPoint4[8267] = {X 367.1193, Y 58.0000, Z -5.5000, A 0.000, B 0.000, C 0.000 }
gfCNCPoint4[8268] = {X 367.2296, Y 57.0209, Z -5.5000, A 0.000, B 0.000, C 0.000 }
gfCNCPoint4[8269] = {X 367.5550, Y 56.0909, Z -5.5000, A 0.000, B 0.000, C 0.000 }
gfCNCPoint4[8270] = {X 368.0792, Y 55.2566, Z -5.5000, A 0.000, B 0.000, C 0.000 }
gfCNCPoint4[8271] = {X 368.7759, Y 54.5599, Z -5.5000, A 0.000, B 0.000, C 0.000 }
gfCNCPoint4[8272] = {X 369.6102, Y 54.0357, Z -5.5000, A 0.000, B 0.000, C 0.000 }
gfCNCPoint4[8273] = {X 370.5402, Y 53.7103, Z -5.5000, A 0.000, B 0.000, C 0.000 }
gfCNCPoint4[8274] = {X 371.5193, Y 53.6000, Z -5.5000, A 0.000, B 0.000, C 0.000 }
gfCNCPoint4[8275] = {X 388.0597, Y 53.6000, Z -5.5000, A 0.000, B 0.000, C 0.000 }
gfCNCPoint4[8276] = {X 389.0388, Y 53.7103, Z -5.5000, A 0.000, B 0.000, C 0.000 }
gfCNCPoint4[8277] = {X 389.9688, Y 54.0357, Z -5.5000, A 0.000, B 0.000, C 0.000 }
gfCNCPoint4[8278] = {X 390.8030, Y 54.5599, Z -5.5000, A 0.000, B 0.000, C 0.000 }
gfCNCPoint4[8279] = {X 391.4997, Y 55.2566, Z -5.5000, A 0.000, B 0.000, C 0.000 }
gfCNCPoint4[8280] = {X 392.0239, Y 56.0909, Z -5.5000, A 0.000, B 0.000, C 0.000 }
gfCNCPoint4[8281] = {X 392.3494, Y 57.0209, Z -5.5000, A 0.000, B 0.000, C 0.000 }
gfCNCPoint4[8282] = {X 392.4597, Y 58.0000, Z -5.5000, A 0.000, B 0.000, C 0.000 }
gfCNCPoint4[8283] = {X 392.4595, Y 58.9704, Z -5.5000, A 0.000, B 0.000, C 0.000 }
gfCNCPoint4[8284] = {X 392.3404, Y 59.9516, Z -5.5000, A 0.000, B 0.000, C 0.000 }
gfCNCPoint4[8285] = {X 392.0053, Y 60.8814, Z -5.5000, A 0.000, B 0.000, C 0.000 }
gfCNCPoint4[8286] = {X 391.5624, Y 61.5976, Z -5.5000, A 0.000, B 0.000, C 0.000 }
gfCNCPoint4[8287] = {X 390.9919, Y 62.2168, Z -5.5000, A 0.000, B 0.000, C 0.000 }
gfCNCPoint4[8288] = {X 390.3143, Y 62.7167, Z -5.5000, A 0.000, B 0.000, C 0.000 }
gfCNCPoint4[8289] = {X 389.5543, Y 63.0792, Z -5.5000, A 0.000, B 0.000, C 0.000 }
gfCNCPoint4[8290] = {X 388.7393, Y 63.2910, Z -5.5000, A 0.000, B 0.000, C 0.000 }
gfCNCPoint4[8291] = {X 388.7393, Y 83.9247, Z -5.5000, A 0.000, B 0.000, C 0.000 }
gfCNCPoint4[8292] = {X 388.7373, Y 84.6150, Z -5.5000, A 0.000, B 0.000, C 0.000 }
gfCNCPoint4[8293] = {X 388.6771, Y 86.2800, Z -5.5000, A 0.000, B 0.000, C 0.000 }
gfCNCPoint4[8294] = {X 388.4719, Y 87.9334, Z -5.5000, A 0.000, B 0.000, C 0.000 }
gfCNCPoint4[8295] = {X 388.1232, Y 89.5627, Z -5.5000, A 0.000, B 0.000, C 0.000 }
gfCNCPoint4[8296] = {X 387.5874, Y 91.1607, Z -5.5000, A 0.000, B 0.000, C 0.000 }
gfCNCPoint4[8297] = {X 386.8327, Y 92.6678, Z -5.5000, A 0.000, B 0.000, C 0.000 }
gfCNCPoint4[8298] = {X 385.8741, Y 94.0542, Z -5.5000, A 0.000, B 0.000, C 0.000 }
gfCNCPoint4[8299] = {X 384.7306, Y 95.2924, Z -5.5000, A 0.000, B 0.000, C 0.000 }
gfCNCPoint4[8300] = {X 383.5026, Y 96.3481, Z -5.5000, A 0.000, B 0.000, C 0.000 }
gfCNCPoint4[8301] = {X 382.1880, Y 97.2936, Z -5.5000, A 0.000, B 0.000, C 0.000 }
gfCNCPoint4[8302] = {X 382.4511, Y 97.6951, Z -5.5000, A 0.000, B 0.000, C 0.000 }
gfCNCPoint4[8303] = {X 391.5259, Y 97.6951, Z -5.5000, A 0.000, B 0.000, C 0.000 }
gfCNCPoint4[8304] = {X 391.5259, Y 97.0659, Z -5.5000, A 0.000, B 0.000, C 0.000 }
gfCNCPoint4[8305] = {X 391.6200, Y 96.1127, Z -5.5000, A 0.000, B 0.000, C 0.000 }
gfCNCPoint4[8306] = {X 391.8983, Y 95.1962, Z -5.5000, A 0.000, B 0.000, C 0.000 }
gfCNCPoint4[8307] = {X 392.3504, Y 94.3518, Z -5.5000, A 0.000, B 0.000, C 0.000 }
gfCNCPoint4[8308] = {X 392.9587, Y 93.6119, Z -5.5000, A 0.000, B 0.000, C 0.000 }
gfCNCPoint4[8309] = {X 393.6998, Y 93.0050, Z -5.5000, A 0.000, B 0.000, C 0.000 }
gfCNCPoint4[8310] = {X 394.5451, Y 92.5546, Z -5.5000, A 0.000, B 0.000, C 0.000 }
gfCNCPoint4[8311] = {X 395.4622, Y 92.2781, Z -5.5000, A 0.000, B 0.000, C 0.000 }
gfCNCPoint4[8312] = {X 396.4156, Y 92.1859, Z -5.5000, A 0.000, B 0.000, C 0.000 }
gfCNCPoint4[8313] = {X 397.3218, Y 92.1441, Z -5.5000, A 0.000, B 0.000, C 0.000 }
gfCNCPoint4[8314] = {X 398.2250, Y 92.0582, Z -5.5000, A 0.000, B 0.000, C 0.000 }
gfCNCPoint4[8315] = {X 398.7530, Y 91.9297, Z -5.5000, A 0.000, B 0.000, C 0.000 }
gfCNCPoint4[8316] = {X 399.2394, Y 91.6872, Z -5.5000, A 0.000, B 0.000, C 0.000 }
gfCNCPoint4[8317] = {X 426.8265, Y 74.0195, Z -5.5000, A 0.000, B 0.000, C 0.000 }
gfCNCPoint4[8318] = {X 403.5509, Y 64.8875, Z -5.5000, A 0.000, B 0.000, C 0.000 }
gfCNCPoint4[8319] = {X 401.9167, Y 64.3462, Z -5.5000, A 0.000, B 0.000, C 0.000 }
gfCNCPoint4[8320] = {X 400.2330, Y 63.9869, Z -5.5000, A 0.000, B 0.000, C 0.000 }
gfCNCPoint4[8321] = {X 398.5202, Y 63.8139, Z -5.5000, A 0.000, B 0.000, C 0.000 }
gfCNCPoint4[8322] = {X 397.5545, Y 63.7098, Z -5.5000, A 0.000, B 0.000, C 0.000 }
gfCNCPoint4[8323] = {X 396.6286, Y 63.4166, Z -5.5000, A 0.000, B 0.000, C 0.000 }
gfCNCPoint4[8324] = {X 395.7791, Y 62.9457, Z -5.5000, A 0.000, B 0.000, C 0.000 }
gfCNCPoint4[8325] = {X 395.0396, Y 62.3160, Z -5.5000, A 0.000, B 0.000, C 0.000 }
gfCNCPoint4[8326] = {X 394.4660, Y 61.5934, Z -5.5000, A 0.000, B 0.000, C 0.000 }
gfCNCPoint4[8327] = {X 394.0386, Y 60.7757, Z -5.5000, A 0.000, B 0.000, C 0.000 }
gfCNCPoint4[8328] = {X 393.7727, Y 59.8921, Z -5.5000, A 0.000, B 0.000, C 0.000 }
gfCNCPoint4[8329] = {X 393.6779, Y 58.9744, Z -5.5000, A 0.000, B 0.000, C 0.000 }
gfCNCPoint4[8330] = {X 393.6777, Y 58.0000, Z -5.5000, A 0.000, B 0.000, C 0.000 }
gfCNCPoint4[8331] = {X 393.7668, Y 57.0718, Z -5.5000, A 0.000, B 0.000, C 0.000 }
gfCNCPoint4[8332] = {X 394.0309, Y 56.1774, Z -5.5000, A 0.000, B 0.000, C 0.000 }
gfCNCPoint4[8333] = {X 394.4602, Y 55.3496, Z -5.5000, A 0.000, B 0.000, C 0.000 }
gfCNCPoint4[8334] = {X 395.0391, Y 54.6186, Z -5.5000, A 0.000, B 0.000, C 0.000 }
gfCNCPoint4[8335] = {X 395.7864, Y 53.9833, Z -5.5000, A 0.000, B 0.000, C 0.000 }
gfCNCPoint4[8336] = {X 396.6455, Y 53.5102, Z -5.5000, A 0.000, B 0.000, C 0.000 }
gfCNCPoint4[8337] = {X 397.5819, Y 53.2186, Z -5.5000, A 0.000, B 0.000, C 0.000 }
gfCNCPoint4[8338] = {X 398.5577, Y 53.1200, Z -5.5000, A 0.000, B 0.000, C 0.000 }
gfCNCPoint4[8339] = {X 419.4886, Y 53.1200, Z -5.5000, A 0.000, B 0.000, C 0.000 }
gfCNCPoint4[8340] = {X 420.5534, Y 53.2376, Z -5.5000, A 0.000, B 0.000, C 0.000 }
gfCNCPoint4[8341] = {X 421.5668, Y 53.5846, Z -5.5000, A 0.000, B 0.000, C 0.000 }
gfCNCPoint4[8342] = {X 422.4801, Y 54.1444, Z -5.5000, A 0.000, B 0.000, C 0.000 }
gfCNCPoint4[8343] = {X 423.2493, Y 54.8900, Z -5.5000, A 0.000, B 0.000, C 0.000 }
gfCNCPoint4[8344] = {X 423.8372, Y 55.7855, Z -5.5000, A 0.000, B 0.000, C 0.000 }
gfCNCPoint4[8345] = {X 424.2156, Y 56.7876, Z -5.5000, A 0.000, B 0.000, C 0.000 }
gfCNCPoint4[8346] = {X 424.3662, Y 57.8482, Z -5.5000, A 0.000, B 0.000, C 0.000 }
gfCNCPoint4[8347] = {X 429.8190, Y 59.9729, Z -5.5000, A 0.000, B 0.000, C 0.000 }
gfCNCPoint4[8348] = {X 457.2984, Y 70.8757, Z -5.5000, A 0.000, B 0.000, C 0.000 }
gfCNCPoint4[8349] = {X 457.2988, Y 63.6740, Z -5.5000, A 0.000, B 0.000, C 0.000 }
gfCNCPoint4[8350] = {X 456.2906, Y 63.3056, Z -5.5000, A 0.000, B 0.000, C 0.000 }
gfCNCPoint4[8351] = {X 455.3874, Y 62.7257, Z -5.5000, A 0.000, B 0.000, C 0.000 }
gfCNCPoint4[8352] = {X 454.6329, Y 61.9623, Z -5.5000, A 0.000, B 0.000, C 0.000 }
gfCNCPoint4[8353] = {X 454.0634, Y 61.0525, Z -5.5000, A 0.000, B 0.000, C 0.000 }
gfCNCPoint4[8354] = {X 453.7066, Y 60.0402, Z -5.5000, A 0.000, B 0.000, C 0.000 }
gfCNCPoint4[8355] = {X 453.5798, Y 58.9744, Z -5.5000, A 0.000, B 0.000, C 0.000 }
gfCNCPoint4[8356] = {X 453.5796, Y 58.0000, Z -5.5000, A 0.000, B 0.000, C 0.000 }
gfCNCPoint4[8357] = {X 453.6734, Y 57.0480, Z -5.5000, A 0.000, B 0.000, C 0.000 }
gfCNCPoint4[8358] = {X 453.9511, Y 56.1325, Z -5.5000, A 0.000, B 0.000, C 0.000 }
gfCNCPoint4[8359] = {X 454.4020, Y 55.2888, Z -5.5000, A 0.000, B 0.000, C 0.000 }
gfCNCPoint4[8360] = {X 455.0089, Y 54.5493, Z -5.5000, A 0.000, B 0.000, C 0.000 }
gfCNCPoint4[8361] = {X 455.7484, Y 53.9424, Z -5.5000, A 0.000, B 0.000, C 0.000 }
gfCNCPoint4[8362] = {X 456.5921, Y 53.4915, Z -5.5000, A 0.000, B 0.000, C 0.000 }
gfCNCPoint4[8363] = {X 457.5076, Y 53.2138, Z -5.5000, A 0.000, B 0.000, C 0.000 }
gfCNCPoint4[8364] = {X 458.4596, Y 53.1200, Z -5.5000, A 0.000, B 0.000, C 0.000 }
gfCNCPoint4[8365] = {X 475.0000, Y 53.1200, Z -5.5000, A 0.000, B 0.000, C 0.000 }
gfCNCPoint4[8366] = {X 475.9520, Y 53.2138, Z -5.5000, A 0.000, B 0.000, C 0.000 }
gfCNCPoint4[8367] = {X 476.8675, Y 53.4915, Z -5.5000, A 0.000, B 0.000, C 0.000 }
gfCNCPoint4[8368] = {X 477.7112, Y 53.9424, Z -5.5000, A 0.000, B 0.000, C 0.000 }
gfCNCPoint4[8369] = {X 478.4507, Y 54.5493, Z -5.5000, A 0.000, B 0.000, C 0.000 }
gfCNCPoint4[8370] = {X 479.0576, Y 55.2888, Z -5.5000, A 0.000, B 0.000, C 0.000 }
gfCNCPoint4[8371] = {X 479.5085, Y 56.1325, Z -5.5000, A 0.000, B 0.000, C 0.000 }
gfCNCPoint4[8372] = {X 479.7862, Y 57.0480, Z -5.5000, A 0.000, B 0.000, C 0.000 }
gfCNCPoint4[8373] = {X 479.8800, Y 58.0000, Z -5.5000, A 0.000, B 0.000, C 0.000 }
gfCNCPoint4[8374] = {X 479.8798, Y 58.9744, Z -5.5000, A 0.000, B 0.000, C 0.000 }
gfCNCPoint4[8375] = {X 479.7530, Y 60.0403, Z -5.5000, A 0.000, B 0.000, C 0.000 }
gfCNCPoint4[8376] = {X 479.3961, Y 61.0526, Z -5.5000, A 0.000, B 0.000, C 0.000 }
gfCNCPoint4[8377] = {X 478.8266, Y 61.9625, Z -5.5000, A 0.000, B 0.000, C 0.000 }
gfCNCPoint4[8378] = {X 478.0720, Y 62.7258, Z -5.5000, A 0.000, B 0.000, C 0.000 }
gfCNCPoint4[8379] = {X 477.1687, Y 63.3057, Z -5.5000, A 0.000, B 0.000, C 0.000 }
gfCNCPoint4[8380] = {X 476.1605, Y 63.6741, Z -5.5000, A 0.000, B 0.000, C 0.000 }
gfCNCPoint4[8381] = {X 476.1609, Y 92.3312, Z -5.5000, A 0.000, B 0.000, C 0.000 }
gfCNCPoint4[8382] = {X 476.3645, Y 92.3909, Z -5.5000, A 0.000, B 0.000, C 0.000 }
gfCNCPoint4[8383] = {X 476.5665, Y 92.4556, Z -5.5000, A 0.000, B 0.000, C 0.000 }
gfCNCPoint4[8384] = {X 477.4837, Y 92.8726, Z -5.5000, A 0.000, B 0.000, C 0.000 }
gfCNCPoint4[8385] = {X 478.2950, Y 93.4701, Z -5.5000, A 0.000, B 0.000, C 0.000 }
gfCNCPoint4[8386] = {X 478.9654, Y 94.2222, Z -5.5000, A 0.000, B 0.000, C 0.000 }
gfCNCPoint4[8387] = {X 479.4661, Y 95.0965, Z -5.5000, A 0.000, B 0.000, C 0.000 }
gfCNCPoint4[8388] = {X 479.7754, Y 96.0554, Z -5.5000, A 0.000, B 0.000, C 0.000 }
gfCNCPoint4[8389] = {X 479.8800, Y 97.0575, Z -5.5000, A 0.000, B 0.000, C 0.000 }
gfCNCPoint4[8390] = {X 479.8800, Y 97.6951, Z -5.5000, A 0.000, B 0.000, C 0.000 }
gfCNCPoint4[8391] = {X 479.4000, Y 97.6951, Z -5.5000, A 0.000, B 0.000, C 0.000 }
gfCNCPoint4[8392] = {X 479.4000, Y 98.0000, Z -5.5000, A 0.000, B 0.000, C 0.000 }
gfCNCPoint4[8393] = {X 479.2897, Y 98.9791, Z -5.5000, A 0.000, B 0.000, C 0.000 }
gfCNCPoint4[8394] = {X 478.9643, Y 99.9091, Z -5.5000, A 0.000, B 0.000, C 0.000 }
gfCNCPoint4[8395] = {X 478.4401, Y 100.7434, Z -5.5000, A 0.000, B 0.000, C 0.000 }
gfCNCPoint4[8396] = {X 477.7434, Y 101.4401, Z -5.5000, A 0.000, B 0.000, C 0.000 }
gfCNCPoint4[8397] = {X 476.9091, Y 101.9643, Z -5.5000, A 0.000, B 0.000, C 0.000 }
gfCNCPoint4[8398] = {X 475.9791, Y 102.2897, Z -5.5000, A 0.000, B 0.000, C 0.000 }
gfCNCPoint4[8399] = {X 475.0000, Y 102.4000, Z -5.5000, A 0.000, B 0.000, C 0.000 }
gfCNCPoint4[8400] = {X 458.4596, Y 102.4000, Z -5.5000, A 0.000, B 0.000, C 0.000 }
gfCNCPoint4[8401] = {X 457.4805, Y 102.2897, Z -5.5000, A 0.000, B 0.000, C 0.000 }
gfCNCPoint4[8402] = {X 456.5505, Y 101.9643, Z -5.5000, A 0.000, B 0.000, C 0.000 }
gfCNCPoint4[8403] = {X 455.7162, Y 101.4401, Z -5.5000, A 0.000, B 0.000, C 0.000 }
gfCNCPoint4[8404] = {X 455.0195, Y 100.7434, Z -5.5000, A 0.000, B 0.000, C 0.000 }
gfCNCPoint4[8405] = {X 454.4953, Y 99.9091, Z -5.5000, A 0.000, B 0.000, C 0.000 }
gfCNCPoint4[8406] = {X 454.1699, Y 98.9791, Z -5.5000, A 0.000, B 0.000, C 0.000 }
gfCNCPoint4[8407] = {X 454.0596, Y 98.0000, Z -5.5000, A 0.000, B 0.000, C 0.000 }
gfCNCPoint4[8408] = {X 454.0596, Y 97.0659, Z -5.5000, A 0.000, B 0.000, C 0.000 }
gfCNCPoint4[8409] = {X 454.1492, Y 96.1826, Z -5.5000, A 0.000, B 0.000, C 0.000 }
gfCNCPoint4[8410] = {X 454.4143, Y 95.3353, Z -5.5000, A 0.000, B 0.000, C 0.000 }
gfCNCPoint4[8411] = {X 454.8440, Y 94.5584, Z -5.5000, A 0.000, B 0.000, C 0.000 }
gfCNCPoint4[8412] = {X 455.4210, Y 93.8836, Z -5.5000, A 0.000, B 0.000, C 0.000 }
gfCNCPoint4[8413] = {X 456.1217, Y 93.3384, Z -5.5000, A 0.000, B 0.000, C 0.000 }
gfCNCPoint4[8414] = {X 456.9176, Y 92.9450, Z -5.5000, A 0.000, B 0.000, C 0.000 }
gfCNCPoint4[8415] = {X 457.7763, Y 92.7193, Z -5.5000, A 0.000, B 0.000, C 0.000 }
gfCNCPoint4[8416] = {X 457.7763, Y 85.6495, Z -5.5000, A 0.000, B 0.000, C 0.000 }
gfCNCPoint4[8417] = {X 444.8685, Y 80.5897, Z -5.5000, A 0.000, B 0.000, C 0.000 }
gfCNCPoint4[8418] = {X 420.1040, Y 96.6316, Z -5.5000, A 0.000, B 0.000, C 0.000 }
gfCNCPoint4[8419] = {X 420.1067, Y 97.0659, Z -5.5000, A 0.000, B 0.000, C 0.000 }
gfCNCPoint4[8420] = {X 420.1067, Y 98.0000, Z -5.5000, A 0.000, B 0.000, C 0.000 }
gfCNCPoint4[8421] = {X 419.9964, Y 98.9791, Z -5.5000, A 0.000, B 0.000, C 0.000 }
gfCNCPoint4[8422] = {X 419.6710, Y 99.9091, Z -5.5000, A 0.000, B 0.000, C 0.000 }
gfCNCPoint4[8423] = {X 419.1468, Y 100.7434, Z -5.5000, A 0.000, B 0.000, C 0.000 }
gfCNCPoint4[8424] = {X 418.4501, Y 101.4401, Z -5.5000, A 0.000, B 0.000, C 0.000 }
gfCNCPoint4[8425] = {X 417.6158, Y 101.9643, Z -5.5000, A 0.000, B 0.000, C 0.000 }
gfCNCPoint4[8426] = {X 416.6858, Y 102.2897, Z -5.5000, A 0.000, B 0.000, C 0.000 }
gfCNCPoint4[8427] = {X 415.7067, Y 102.4000, Z -5.5000, A 0.000, B 0.000, C 0.000 }
gfCNCPoint4[8428] = {X 396.4059, Y 102.4000, Z -5.5000, A 0.000, B 0.000, C 0.000 }
gfCNCPoint4[8429] = {X 395.4269, Y 102.2897, Z -5.5000, A 0.000, B 0.000, C 0.000 }
gfCNCPoint4[8430] = {X 394.4969, Y 101.9643, Z -5.5000, A 0.000, B 0.000, C 0.000 }
gfCNCPoint4[8431] = {X 393.6626, Y 101.4401, Z -5.5000, A 0.000, B 0.000, C 0.000 }
gfCNCPoint4[8432] = {X 392.9659, Y 100.7434, Z -5.5000, A 0.000, B 0.000, C 0.000 }
gfCNCPoint4[8433] = {X 392.4417, Y 99.9091, Z -5.5000, A 0.000, B 0.000, C 0.000 }
gfCNCPoint4[8434] = {X 392.1163, Y 98.9791, Z -5.5000, A 0.000, B 0.000, C 0.000 }
gfCNCPoint4[8435] = {X 392.0059, Y 98.0000, Z -5.5000, A 0.000, B 0.000, C 0.000 }
gfCNCPoint4[8436] = {X 392.0059, Y 97.0659, Z -5.5000, A 0.000, B 0.000, C 0.000 }
gfCNCPoint4[8437] = {X 392.1167, Y 96.0849, Z -5.5000, A 0.000, B 0.000, C 0.000 }
gfCNCPoint4[8438] = {X 392.4434, Y 95.1532, Z -5.5000, A 0.000, B 0.000, C 0.000 }
gfCNCPoint4[8439] = {X 392.9697, Y 94.3178, Z -5.5000, A 0.000, B 0.000, C 0.000 }
gfCNCPoint4[8440] = {X 393.6689, Y 93.6208, Z -5.5000, A 0.000, B 0.000, C 0.000 }
gfCNCPoint4[8441] = {X 394.5060, Y 93.0973, Z -5.5000, A 0.000, B 0.000, C 0.000 }
gfCNCPoint4[8442] = {X 395.4387, Y 92.7736, Z -5.5000, A 0.000, B 0.000, C 0.000 }
gfCNCPoint4[8443] = {X 396.4201, Y 92.6660, Z -5.5000, A 0.000, B 0.000, C 0.000 }
gfCNCPoint4[8444] = {X 397.3536, Y 92.6230, Z -5.5000, A 0.000, B 0.000, C 0.000 }
gfCNCPoint4[8445] = {X 398.2838, Y 92.5346, Z -5.5000, A 0.000, B 0.000, C 0.000 }
gfCNCPoint4[8446] = {X 398.9171, Y 92.3808, Z -5.5000, A 0.000, B 0.000, C 0.000 }
gfCNCPoint4[8447] = {X 399.5003, Y 92.0901, Z -5.5000, A 0.000, B 0.000, C 0.000 }
gfCNCPoint4[8448] = {X 405.1764, Y 88.4328, Z -5.5000, A 0.000, B 0.000, C 0.000 }
gfCNCPoint4[8449] = {X 427.8785, Y 73.9166, Z -5.5000, A 0.000, B 0.000, C 0.000 }
gfCNCPoint4[8450] = {X 403.7262, Y 64.4406, Z -5.5000, A 0.000, B 0.000, C 0.000 }
gfCNCPoint4[8451] = {X 402.0391, Y 63.8821, Z -5.5000, A 0.000, B 0.000, C 0.000 }
gfCNCPoint4[8452] = {X 400.3010, Y 63.5117, Z -5.5000, A 0.000, B 0.000, C 0.000 }
gfCNCPoint4[8453] = {X 398.5328, Y 63.3340, Z -5.5000, A 0.000, B 0.000, C 0.000 }
gfCNCPoint4[8454] = {X 397.5578, Y 63.2189, Z -5.5000, A 0.000, B 0.000, C 0.000 }
gfCNCPoint4[8455] = {X 396.6326, Y 62.8906, Z -5.5000, A 0.000, B 0.000, C 0.000 }
gfCNCPoint4[8456] = {X 395.8032, Y 62.3652, Z -5.5000, A 0.000, B 0.000, C 0.000 }
gfCNCPoint4[8457] = {X 395.1110, Y 61.6690, Z -5.5000, A 0.000, B 0.000, C 0.000 }
gfCNCPoint4[8458] = {X 394.5904, Y 60.8367, Z -5.5000, A 0.000, B 0.000, C 0.000 }
gfCNCPoint4[8459] = {X 394.2672, Y 59.9097, Z -5.5000, A 0.000, B 0.000, C 0.000 }
gfCNCPoint4[8460] = {X 394.1577, Y 58.9341, Z -5.5000, A 0.000, B 0.000, C 0.000 }
gfCNCPoint4[8461] = {X 394.1577, Y 58.0000, Z -5.5000, A 0.000, B 0.000, C 0.000 }
gfCNCPoint4[8462] = {X 394.2680, Y 57.0209, Z -5.5000, A 0.000, B 0.000, C 0.000 }
gfCNCPoint4[8463] = {X 394.5935, Y 56.0909, Z -5.5000, A 0.000, B 0.000, C 0.000 }
gfCNCPoint4[8464] = {X 395.1177, Y 55.2566, Z -5.5000, A 0.000, B 0.000, C 0.000 }
gfCNCPoint4[8465] = {X 395.8144, Y 54.5599, Z -5.5000, A 0.000, B 0.000, C 0.000 }
gfCNCPoint4[8466] = {X 396.6486, Y 54.0357, Z -5.5000, A 0.000, B 0.000, C 0.000 }
gfCNCPoint4[8467] = {X 397.5786, Y 53.7103, Z -5.5000, A 0.000, B 0.000, C 0.000 }
gfCNCPoint4[8468] = {X 398.5577, Y 53.6000, Z -5.5000, A 0.000, B 0.000, C 0.000 }
gfCNCPoint4[8469] = {X 419.4886, Y 53.6000, Z -5.5000, A 0.000, B 0.000, C 0.000 }
gfCNCPoint4[8470] = {X 420.4677, Y 53.7103, Z -5.5000, A 0.000, B 0.000, C 0.000 }
gfCNCPoint4[8471] = {X 421.3977, Y 54.0357, Z -5.5000, A 0.000, B 0.000, C 0.000 }
